// TwinCAT 3 PLC project PLC
// ProgramVersion: 3.1.4024.0
// CompilerDefines: VISU_USEWSTRING
// libraries:
//   CmpBitmapPool, * (System)
//   VisuElemBase, * (System)
//   Tc2_Standard, * (Beckhoff Automation GmbH)
//   Tc2_System, * (Beckhoff Automation GmbH)
//   Tc2_Utilities, * (Beckhoff Automation GmbH)
//   Tc3_Module, * (Beckhoff Automation GmbH)
//   VisuDialogs, * (System)
//   VisuUserMgmt, * (System)
//   VisuSymbols,3.5.10.0,System
//   VisuUserMgmt3 Interfaces,newest,System
// project tree:
//   DUTs/DUTs/DUTs/DUTs_Events/ ST_EventDefinition.TcDUT, ST_EventHistoricalSimple.TcDUT, ST_EventHistoricalSimplePersistent.TcDUT
//   DUTs/DUTs/DUTs/DUTs_HMI/ stButton.TcDUT
//   DUTs/ E_AI_Status.TcDUT, E_Mode.TcDUT
//   / GlobalTextList.TcGTLO, PlcTask.TcTTO
//   GVLs/ GVL.TcGVL, GVL_ForceMode.TcGVL, GVL_IO.TcGVL
//   GVLs/GVLs/GVLs/GVLs_Events/ GVL_EHS.TcGVL, GVL_EHSP.TcGVL, GVL_Event.TcGVL
//   GVLs/GVLs_1/ GVL_Recipe.TcGVL
//   HMI/DUTs_HMI/ stButton_1.TcDUT
//   HMI/FB/ FB_Blink_S.TcPOU, HMI.TcPOU
//   HMI/ GVL_HMI.TcGVL
//   HMI/ListyTextowe/ PrzyciskAlarmy.TcTLO, Tensometr.TcTLO, TextList_Przyciski_Menu.TcTLO
//   HMI/NEW_VISU/Frames/ E0.TcVIS, E1.TcVIS, E2.TcVIS
//   HMI/NEW_VISU/ MAIN.TcVIS, MENU_2.TcVIS, TOP.TcVIS
//   POUs/ Alarms.TcPOU, BreakthroughDetection_2.TcPOU, HydraulicPump.TcPOU, IO_Map.TcPOU, MAIN.TcPOU, Mode.TcPOU, Scaling.TcPOU, UpperPreserDrive.TcPOU, SavePresistent.TcPOU
//   POUs/FB/ FB_4_20mA_To_0_10V.TcPOU, FB_AI_Int_To_PV.TcPOU, FB_AI_mA_To_mm_Adv.TcPOU, FB_AI_Real_To_PV_Adv.TcPOU, FB_AutoManual.TcPOU, FB_Blink_S_1.TcPOU, FB_HydraulicPress_Atos_420mA.TcPOU, FB_HydraulicPumpControl.TcPOU, FB_LongPressLatch.TcPOU, FB_PositionOffset_4_20mA.TcPOU, FB_PressureToForce_PT1.TcPOU, FB_PV_To4_20mA.TcPOU, FB_RevMotorControl.TcPOU, FB_ScaleStrainGaugeForce.TcPOU, FB_ScaleTo0_10V.TcPOU, FB_ScaleTo4_20mA.TcPOU, FB_HydraulicPress_WithBreakthroughDetection_1.TcPOU
//   POUs/POUs/Events/ F_RESET_Event.TcPOU, F_SET_Event.TcPOU, P_EventHandling2.TcPOU, P_Events.TcPOU, P_EventsDefinition.TcPOU, P_EventsHandling.TcPOU, P_EventsVisu.TcPOU
//   POUs/POUs/Recipe/ RecipeManagement.TcPOU
//   VISUs/ Visualization Manager.TcVMO (not stored)
//   VISUs/VISUs/ VISU_TASK.TcTTO
// real-time tasks:
//   TASK PlcTask: cycle T#10ms, priority 20, ADS port 350
//   TASK VISU_TASK: cycle T#200000us, priority 30, ADS port 351
// I/O:
//   DEVICE Device 1 (EtherCAT) (disabled), AmsNetId 192.168.1.80.2.1
//     Term 1 (EK1818) [EK1818 EtherCAT IO-Coupler  (1A E-Bus, 8 Ch. Dig. In, 3ms, 4 Ch. Dig. Out 24V, 0,5A)]
//       Term 2 (EL4374) [EL4374 2Ch. Ana. Input, 2Ch. Ana. Output, +/-10V, +/-20mA, 16 Bit]
//       Term 6 (EL3064) [EL3064 4Ch. Ana. Input 0-10V]
//       Term 3 (EL1008) [EL1008 8Ch. Dig. Input 24V, 3ms]
//       Term 4 (EL2008) [EL2008 8Ch. Dig. Output 24V, 0.5A]
//       Term 5 (EL9011) [EL9011 End Terminal]
// variable links:
//   PLC/PLC Instance <-> Device 1 (EtherCAT)/Term 1 (EK1818)
//     PlcTask Inputs/GVL_IO.DI1_{1..8} <-> Channel {1..8}/GVL_IO.DI1_{1..8}  (8 links)
//     PlcTask Outputs/GVL_IO.DO1_{1..4} <-> Channel {9..12}/Output  (4 links)
//   PLC/PLC Instance <-> Device 1 (EtherCAT)/Term 1 (EK1818)/Term 2 (EL4374)
//     PlcTask Inputs/GVL_IO.AI_1 <-> AI Standard (Real32) Ch.1/GVL_IO.AI_1
//     PlcTask Inputs/GVL_IO.AI_2 <-> AI Standard (Real32) Ch.2/GVL_IO.AI_2
//     PlcTask Outputs/GVL_IO.AO_1 <-> AO Standard (Real32) Ch.3/GVL_IO.AO_1
//   PLC/PLC Instance <-> Device 1 (EtherCAT)/Term 1 (EK1818)/Term 3 (EL1008)
//     PlcTask Inputs/GVL_IO.DI2_{1..8} <-> Channel {1..8}/GVL_IO.DI2_{1..8}  (8 links)
//   PLC/PLC Instance <-> Device 1 (EtherCAT)/Term 1 (EK1818)/Term 4 (EL2008)
//     PlcTask Outputs/GVL_IO.DO2_{1..8} <-> Channel {1..8}/GVL_IO.DO2_{1..8}  (8 links)

CONFIGURATION PLC
    RESOURCE PLC ON TwinCAT3
        TASK PlcTask(INTERVAL := T#10ms, PRIORITY := 20);
        TASK VISU_TASK(INTERVAL := T#200000us, PRIORITY := 30);
        PROGRAM MAIN WITH PlcTask : MAIN;
        PROGRAM VisuElems_Visu_Prg WITH VISU_TASK : VisuElems.Visu_Prg;
    END_RESOURCE
END_CONFIGURATION

// ---- DUTs/DUTs/DUTs/DUTs_Events/ST_EventDefinition.TcDUT
//==================================================================================================
//							Beckhoff Automation Poland
//									23.05.2017
//	Struktura zawierajaca definicje zdarzenia
// 	v1.0	|| TC v 3.1.4020.32		|| - pierwsza wersja
//==================================================================================================
TYPE ST_EventDefinition :
STRUCT
	dwClass									: DWORD;
	dwParam									: DWORD;
	wsMessage								: WSTRING(80);
	bActive									: BOOL;	
END_STRUCT
END_TYPE

// ---- DUTs/DUTs/DUTs/DUTs_Events/ST_EventHistoricalSimple.TcDUT
//==================================================================================================
//							Beckhoff Automation Poland
//									23.05.2017
//	Struktura zawierajaca zdarzenie - pelne informacje, np. do wizualizacji
// 	v1.0	|| TC v 3.1.4020.32		|| - pierwsza wersja
//==================================================================================================
TYPE ST_EventHistoricalSimple :
STRUCT
	dwID									: DWORD;
	dwParam									: DWORD;
	dwClass									: DWORD;
	dtDateBegin								: STRING(19);//DT;
	dtDateEnd								: STRING(19);//DT;
	wsMessage								: WSTRING(80);
	dwColor									: UDINT;
END_STRUCT
END_TYPE

// ---- DUTs/DUTs/DUTs/DUTs_Events/ST_EventHistoricalSimplePersistent.TcDUT
//==================================================================================================
//							Beckhoff Automation Poland
//									23.05.2017
//	Struktura zawierajaca zane do przechowania zdarzenia w pamieci
// 	v1.0	|| TC v 3.1.4020.32		|| - pierwsza wersja
//==================================================================================================
TYPE ST_EventHistoricalSimplePersistent :
STRUCT
	dwID									: DWORD;
	dwParam									: DWORD;
	dwClass									: DWORD;
	dtDateBegin								: STRING(19);//DT;
	dtDateEnd								: STRING(19);//DT;
END_STRUCT
END_TYPE

// ---- DUTs/DUTs/DUTs/DUTs_HMI/stButton.TcDUT
TYPE stButton :
STRUCT
	{attribute 'TcEncoding':='UTF-8'}
	sName				: T_MaxString;
	bToggleCollor		: BOOL;
	bVisable			: BOOL;
	nIndexDynamicText	: UINT;
	dwColor				: DWORD;
	dwAlarmColor		: DWORD;
	
END_STRUCT
END_TYPE

// ---- DUTs/E_AI_Status.TcDUT
//{attribute 'qualified_only'}
//{attribute 'strict'}
TYPE E_AI_Status  :
(
	 AI_Status_Ok,           // wszystko w normie
    AI_Status_UnderRange,   // prąd poniżej dolnego progu (np. przerwana pętla)
    AI_Status_OverRange,    // prąd powyżej górnego progu (np. zwarcie, błąd)
    AI_Status_ConfigError   // błąd konfiguracji (InMin/InMax)
);
END_TYPE

// ---- DUTs/E_Mode.TcDUT
//{attribute 'qualified_only'}
//{attribute 'strict'}
TYPE E_Mode :
(
	Mode_Manual := 0,
    Mode_Auto   := 1
);
END_TYPE

// ---- HMI/DUTs_HMI/stButton_1.TcDUT
TYPE stButton_1 :
STRUCT
	{attribute 'TcEncoding':='UTF-8'}
	sName				: T_MaxString;
	bToggleCollor		: BOOL;
	bVisable			: BOOL;
	nIndexDynamicText	: UINT;
	dwColor				: DWORD;
	dwAlarmColor		: DWORD;
	
END_STRUCT
END_TYPE

// ---- GVLs/GVL.TcGVL
//{attribute 'qualified_only'}
VAR_GLOBAL
	AlwaysFalse					:BOOL;
	
	bControlOn					: BOOL;//kluczyk-sterowanie załączone
	bTopPreserCmdUp				: BOOL;//przycisk kolumna dociskowa do góry
	bTopPreserCmdDown			: BOOL;//przycisk kolumna dociskowa do dołu
	bCycleStartCmd				: BOOL;//przycisk start cyklu
	bCycleStopCmd				: BOOL;//przycisk stop cyklu
	bCylinderCmdUp				: BOOL;//przycisk siłownik do góry
	bCylinderCmdDown			: BOOL;//przycisk siłownik do góry
	bHydraulicUnitCmdStart		: BOOL;//przycisk agregat hydrauliczny start
	nHydraulicPressureRaw		: REAL;//ciśnienie hydrauliki-wejście analogowe
	nCylinderPositionRaw		: REAL;//pozycja siłownika-wejście analogowe
	nHydraulicPressureOut		: REAL;//cisnienie zadane na wyjscie analogowe
	bHydraulicUnitOn			: BOOL;//pottwierdzenie załączenia silnika hydrauliki z softstart
	bTopPreserClosed			: BOOL;//potwierdzenie zamknięcia docisku górnego
	bTopPreserMotorOk			: BOOL;//termik silnika docisku górnego
	bHydraulicUnitMotorOk		: BOOL;//termik silnika hydrauliki
	bHydraulicUnitCmdStop		: BOOL;//przycisk agregat hydrauliczny stop
	bOilLevelOk					: BOOL;//poziom oleju	
	bHydraulicUnitRunning       : BOOL;//softstart hydrauliki załączony
	
	bTopPreserUp				: BOOL;// wyjście -docisk górny do góry
	bTopPreserDown				: BOOL;// wyjście -docisk górny do dołu
	bHydraulicUintOn			: BOOL;// wyjście -załączenie agregatu hydraulicznego
	bLedCycleOn					: BOOL;// wyjście -LED cykl załączony
	bReliefValveOn				: BOOL;// wyjście -zawór odciążający załączony
	bCylinderValveUp			: BOOL;// wyjście -zawór siłownik do góry
	bCylinderValveDown			: BOOL;// wyjście -zawór siłownik do dołu
	bProportionalValveEnable	: BOOL;// wyjście -zawór proporcjonalny załączony	
	bLedHydraulicUnitOn			: BOOL;// wyjście -LED hydraulika załączona
	
	
	

	nHydraulicPressureOut0_10V: LREAL;
END_VAR

// ---- GVLs/GVLs/GVLs/GVLs_Events/GVL_EHS.TcGVL
//==================================================================================================
//							Beckhoff Automation Poland
//									23.05.2017
// 	v1.0	|| TC v 3.1.4020.32		|| - pierwsza wersja
//==================================================================================================
{attribute 'qualified_only'}
VAR_GLOBAL CONSTANT
	diEventsDefinition						: UDINT 	:= 1000;				// Rozmiar tablicy definicji zdarzen, powinna byc w zakresie 5..1000
	diNoOfEvents							: UDINT 	:= 1000;				// Rozmiar tablicy zdarzen historycznych, powinna byc w zakresie 5..1000
END_VAR
VAR_GLOBAL
	stActTime								: TIMESTRUCT;				// Aktualny czas sytemowy w formie struktury
	dtActTime								: STRING(19);//DT;						// Aktualny czas sytemowy
	arrEventDefinition 						: ARRAY [1..GVL_EHS.diEventsDefinition] OF ST_EventDefinition;
	arrEventVisu							: ARRAY [1..GVL_EHS.diNoOfEvents] OF ST_EventHistoricalSimple;		// Pokazywane na wizualizacji - po filtracji
	dwLanguageId							: DWORD := 1045;			// Kod jezyka wyswietlania - Microsoft Locale ID Values
END_VAR

// ---- GVLs/GVLs/GVLs/GVLs_Events/GVL_EHSP.TcGVL
//==================================================================================================
//							Beckhoff Automation Poland
//									23.05.2017
// 	v1.0	|| TC v 3.1.4020.32		|| - pierwsza wersja
//==================================================================================================
{attribute 'qualified_only'}
VAR_GLOBAL PERSISTENT
	arrEvent								: ARRAY [1..GVL_EHS.diNoOfEvents] OF ST_EventHistoricalSimplePersistent;
END_VAR

// ---- GVLs/GVLs/GVLs/GVLs_Events/GVL_Event.TcGVL
{attribute 'qualified_only'}
VAR_GLOBAL
	bAlarm :BOOL;
	bWarning:BOOL;
	bMessage:BOOL;
	aAlarm: ARRAY[0..100] OF BOOL;
	aWarning: ARRAY[0..100] OF BOOL;
	aMessage: ARRAY[0..100] OF BOOL;
	bJestAalrm: BOOL;
	bFilterActiveOnly2: BOOL;
	bJestOstrzezenie: BOOL;
	bJestAalrmLekki: BOOL;
END_VAR

// ---- GVLs/GVLs_1/GVL_Recipe.TcGVL
{attribute 'qualified_only'}
VAR_GLOBAL CONSTANT
	cMaxTableRows 			: INT := 30;

END_VAR
VAR_GLOBAL
	// zmienne receptury
	(*Zmienna1				: LREAL;
	Zmienna2				: LREAL;
	Zmienna3				: LREAL;
	Zmienna4				: LREAL;
	Zmienna5				: INT;
	Zmienna6				: INT;
	Zmienna7				: LREAL;
	Zmienna8				: LREAL;
	Zmienna9				: LREAL;
	Zmienna10				: LREAL;
	*)
	// zmienne do obslugi
	nRecipeCount			: INT;
	aRecipeNames 			: ARRAY[0..cMaxTableRows] OF STRING;
	aVariableNames 			: ARRAY[0..cMaxTableRows] OF STRING;
	aVariableValues 		: ARRAY[0..cMaxTableRows] OF STRING;
	nRecipeIndex			: INT;
	nRecipeSelectionIndex	: INT;
	nVariableIndex			: INT;
	aCurrentValues			: ARRAY[0..cMaxTableRows] OF LREAL;
	


	bZapiszParametry: BOOL;
	bCzytajParametry: BOOL;
	nRecipeSelectionIndexTemp: INT;
	
END_VAR

// ---- GVLs/GVL_ForceMode.TcGVL
{attribute 'qualified_only'}
VAR_GLOBAL
(* ===== Przełączniki =====
	   bModeForce:        FALSE = regulacja i przebicie od ciśnienia (jak dotychczas)
	                      TRUE  = regulacja i przebicie od siły
	   bForceRange100t:   FALSE = tensometr 50 t  (2,5 V = 50 t)
	                      TRUE  = tensometr 100 t (2,5 V = 100 t)
	   Oba można podpiąć pod przełącznik na pulpicie albo pod HMI.
	   Domyślnie FALSE, więc po wgraniu maszyna zostaje w trybie ciśnienia, zakres 50 t.
	*)
	bModeForce					: BOOL := FALSE;
	bForceRange100t				: BOOL := FALSE;

	(* ===== Drugi setpoint — siła [t] =====
	   Odpowiednik setpointów ciśnienia. Używane tylko w trybie siły.
	   Wartość wpisana powyżej wybranego zakresu jest obcinana (patrz *_Eff).
	*)
	nForceSetpointManual		: REAL := 0.0;	(* t, tryb ręczny *)
	nForceSetpointAutoMin		: REAL := 0.0;	(* t, auto *)
	nForceSetpointAutoMax		: REAL := 0.0;	(* t, auto *)
	nBreakDeltaForce			: REAL := 0.0;	(* t, spadek siły w oknie czasu = przebicie *)

	(* ===== Pomiar =====
	   Powiąż nForceInput_V z kanałem AI 0–10 V. Jednostka: wolty (0.0 … 10.0).
	   Zakres roboczy przetwornika to 0.0 … 2.5 V. Powyżej 2.55 V = błąd zakresu.
	*)
	nForceInput_V				: REAL := 0.0;

	nForce_t					: REAL;	(* wartość chwilowa, t *)
	nForce_kg					: REAL;	(* kgf *)
	nForce_N					: REAL;
	nForce_kN					: REAL;
	nForce_pct					: REAL;	(* % wybranego zakresu *)
	nForceFullScale_t			: REAL;	(* 50 albo 100 *)
	bForceSensorOk				: BOOL;
	bForceOverrange				: BOOL;
	bForceUnderrange			: BOOL;

	nForce_Target				: REAL;	(* bieżące zadanie siły w trybie siły [t]; 0 w trybie ciśnienia *)

	

	(* Setpointy faktycznie podane do regulatora po obcięciu do zakresu. *)
	nForceSetpointManual_Eff	: REAL;
	nForceSetpointAutoMin_Eff	: REAL;
	nForceSetpointAutoMax_Eff	: REAL;
	nBreakDeltaForce_Eff		: REAL;
	bForceSetpointLimited		: BOOL;	(* wpisana wartość była poza 0 … pełny zakres albo delta < 0 *)
	bForceCfgFault				: BOOL;	(* AutoMin > AutoMax po obcięciu *)
	bForceInhibit				: BOOL;	(* tryb siły i zły tensometr — ruch w górę jest zablokowany, dół zostaje *)
	bMotionHold					: BOOL;	(* zmiana trybu lub zakresu 50/100 t w ruchu — puść przyciski *)
	bRegulatorActive			: BOOL;
	bAlarm						: BOOL;
	nActiveSetpointManual		: REAL;	(* to, co w tym cyklu poszło jako setpoint ręczny: bar albo t *)
	nActiveActual				: REAL;	(* to, co w tym cyklu poszło jako wartość rzeczywista *)
END_VAR

// ---- GVLs/GVL_IO.TcGVL
//{attribute 'qualified_only'}
VAR_GLOBAL
//---------------------------------------------	
// EK 1818

	DI1_1 AT %I*: BOOL;
	DI1_2 AT %I*: BOOL;
	DI1_3 AT %I*: BOOL;
	DI1_4 AT %I*: BOOL;
	DI1_5 AT %I*: BOOL;
	DI1_6 AT %I*: BOOL;
	DI1_7 AT %I*: BOOL;
	DI1_8 AT %I*: BOOL;
	
	DO1_1 AT %Q*: BOOL;
	DO1_2 AT %Q*: BOOL;
	DO1_3 AT %Q*: BOOL;
	DO1_4 AT %Q*: BOOL;
//--------------------------------------------	
// EL 4374	
	AI_1 AT %I*: REAL;
	AI_2 AT %I*: REAL;
	AO_1 AT %Q*: REAL;
	AO_2 AT %Q*: REAL;
//--------------------------------------------
// EL 1008	
	DI2_1 AT %I*: BOOL;
	DI2_2 AT %I*: BOOL;
	DI2_3 AT %I*: BOOL;
	DI2_4 AT %I*: BOOL;
	DI2_5 AT %I*: BOOL;
	DI2_6 AT %I*: BOOL;
	DI2_7 AT %I*: BOOL;
	DI2_8 AT %I*: BOOL;
	
//--------------------------------------------
//EL 2008
	DO2_1 AT %Q*: BOOL;
	DO2_2 AT %Q*: BOOL;
	DO2_3 AT %Q*: BOOL;
	DO2_4 AT %Q*: BOOL;
	DO2_5 AT %Q*: BOOL;
	DO2_6 AT %Q*: BOOL;
	DO2_7 AT %Q*: BOOL;
	DO2_8 AT %Q*: BOOL;
	// sygnał z przekaźnika bezpieczeństwa
	bEstopOk: BOOL;
END_VAR

// ---- HMI/GVL_HMI.TcGVL
{attribute 'qualified_only'}
VAR_GLOBAL
	hmiPanel	: HMI;
	
	bKlodka: BOOL;
	bResetAlarm: BOOL;
	
	tBreak_Time_Window: TIME;
	sMode: STRING;
	nPressBreak: REAL;
	nPositionBreak: REAL;
	nPressStart: REAL;
	nPositionStart: REAL;
	Force_N: REAL;
	Force_kg: REAL;
	Force_kg_2: REAL;
	Force_N_2: REAL;
	(* Zatrzask w chwili wykrycia przebicia — pomiar z tensometru, niezależnie od trybu. *)
	nForce_t_Break				: REAL;
	nForce_kg_Break				: REAL;
	nForce_N_Break				: REAL;
	nForce_kN_Break				: REAL;
END_VAR
VAR_GLOBAL PERSISTENT
	nBreak_Time_Window			: INT;
	nPressureSetpointManual: REAL;
	nBreakDeltaPress: REAL;
	nBreakDeltaPos: REAL;
	PressureSetpointAutoMin: LREAL;
	PressureSetpointAutoMax: LREAL;
	// czas rampy Auto[ms]
	nRamp_Time: DINT:=120;
END_VAR
VAR_GLOBAL CONSTANT
	// Czasem w HMI trzeba podać kolor w wersji 16 
	dwRed				: DWORD  := 16#FFE62545;
	dwGreen				: DWORD  := 16#FF007D00;
	dwYelow				: DWORD  := 16#FFFFFF00;
	dwBlack				: DWORD  := 16#FF000000;
	dwGrey_B			: DWORD  := 16#FF636363;
	dwGrey_W			: DWORD  := 16#FFC8C8C8;
	dwWhite				: DWORD  := 16#FFFFFFFF;
	dwBackGround		: DWORD	 := 16#FFABA494;
	
END_VAR

// ---- POUs/MAIN.TcPOU
PROGRAM MAIN
VAR
END_VAR

GVL_HMI.hmiPanel();

UpperPreserDrive();
HydraulicPump();
BreakthroughDetection_2();



P_Events();
P_EventsDefinition();
Alarms();
Scaling();
SavePresistent();
Mode();
IO_Map();

END_PROGRAM

// ---- POUs/UpperPreserDrive.TcPOU
PROGRAM UpperPreserDrive
VAR
	fbUupperPreser: FB_RevMotorControl;
	
	bStop: BOOL;
	
END_VAR

fbUupperPreser(
	bForward:=.bTopPreserCmdDown , 
	bReverse:=.bTopPreserCmdUp , 
	bStop:=bStop , 
	bThermalOk:=.bTopPreserMotorOk , 
	bLimitSwitchFwd:=TRUE , 
	bLimitSwitchRev:=.bTopPreserClosed , 
	bEmergencyStop:=.bEstopOk , 
	bEnable:=bControlOn , 
	bRunForward=>.bTopPreserDown , 
	bRunReverse=>.bTopPreserUp , 
	bRunning=> , 
	bFault=> , 
	bReady=> );

END_PROGRAM

// ---- POUs/FB/FB_RevMotorControl.TcPOU
FUNCTION_BLOCK FB_RevMotorControl
VAR_INPUT
    bForward            : BOOL;  // Komenda jazdy w przód
    bReverse            : BOOL;  // Komenda jazdy w tył
    bStop               : BOOL := FALSE;  // Zatrzymanie ręczne (opcjonalne)
    bThermalOk          : BOOL := TRUE;   // Termik silnika OK (NC → 0 = zadziałany)
    bLimitSwitchFwd     : BOOL := TRUE;   // Krańcówka przód (NC → 0 = osiągnięta)
    bLimitSwitchRev     : BOOL := TRUE;   // Krańcówka tył  (NC → 0 = osiągnięta)
    bEmergencyStop      : BOOL := TRUE;   // E-Stop (NC → 0 = wciśnięty)
    bEnable             : BOOL := TRUE;   // Zewnętrzne zezwolenie
END_VAR

VAR_OUTPUT
    bRunForward         : BOOL;  // Stycznik – jazda w przód
    bRunReverse         : BOOL;  // Stycznik – jazda w tył
    bRunning            : BOOL;  // Silnik pracuje (którykolwiek kierunek)
    bFault              : BOOL;  // Błąd wymagający kasowania (głównie termik)
    bReady              : BOOL;  // System gotowy do pracy
END_VAR

VAR
    bIntForward         : BOOL := FALSE;  // Wewnętrzny stan przód
    bIntReverse         : BOOL := FALSE;  // Wewnętrzny stan tył
    bThermalFault       : BOOL := FALSE;  // Ręczna pamięć błędu termicznego (zamiast SR)
    tAntiTieDelay1       : TON;            // Opóźnienie przeciwzwarciowe 400 ms
	tAntiTieDelay2       : TON;            // Opóźnienie przeciwzwarciowe 400 ms
    bFirstCycle         : BOOL := TRUE;
END_VAR



//===================================================================
// Poprawiona logika – krańcówki działają prawidłowo!
//===================================================================

IF bFirstCycle THEN
  
    tAntiTieDelay1.PT := T#300MS;
	tAntiTieDelay2.PT := T#300MS;
	  bFirstCycle := FALSE;
END_IF;

// 1. Natychmiastowe wyłączenie przy braku bezpieczeństwa
IF NOT bEmergencyStop OR NOT bThermalOk THEN
    bIntForward := FALSE;
    bIntReverse := FALSE;
END_IF;

// 2. Ręczna pamięć błędu termicznego
IF NOT bThermalOk AND bRunForward AND bRunReverse THEN
    bThermalFault := TRUE;                    // SET
END_IF;
IF bEmergencyStop AND bThermalOk AND (bStop OR (bForward AND bReverse)) THEN
    bThermalFault := FALSE;                   // RST
END_IF;

// 3. Główna logika kierunku – KRAŃCÓWKI TYLKO BLOKUJĄ SWÓJ KIERUNEK!
IF NOT bThermalFault AND bEnable AND bEmergencyStop AND bThermalOk THEN

    // Żądanie jazdy w przód – dozwolone tylko jeśli krańcówka przód jest zwolniona
    IF bForward AND NOT bReverse AND bLimitSwitchFwd AND NOT bIntReverse THEN
        bIntForward := TRUE;
    ELSIF NOT bLimitSwitchFwd OR bReverse THEN
        bIntForward := FALSE;                 // krańcówka przód osiągnięta → wyłącz przód
    END_IF;

    // Żądanie jazdy w tył – dozwolone tylko jeśli krańcówka tył jest zwolniona
    IF bReverse AND NOT bForward AND bLimitSwitchRev and not bIntForward THEN
        bIntReverse := TRUE;
    ELSIF NOT bLimitSwitchRev OR bForward THEN
        bIntReverse := FALSE;                 // krańcówka tył osiągnięta → wyłącz tył
    END_IF;

    // Zatrzymanie ręczne lub brak komendy
    IF bStop OR (NOT bForward AND NOT bReverse)OR (bForward AND  bReverse) THEN
        bIntForward := FALSE;
        bIntReverse := FALSE;
    END_IF;

END_IF;

// 4. Opóźnienie przeciwzwarciowe 400 ms
tAntiTieDelay1(IN := bForward );

IF tAntiTieDelay1.Q THEN
    bRunForward := bIntForward;
    
ELSE
    bRunForward := FALSE;
   
END_IF;

tAntiTieDelay2(IN := bReverse);

IF tAntiTieDelay2.Q THEN
   
    bRunReverse := bIntReverse;
ELSE
   
    bRunReverse := FALSE;
END_IF;
// 5. Wyjścia diagnostyczne
bRunning := bRunForward OR bRunReverse;

bReady   := bEmergencyStop
            AND bThermalOk
            AND bEnable
            AND NOT bThermalFault;

bFault   := bThermalFault;

END_FUNCTION_BLOCK

// ---- POUs/HydraulicPump.TcPOU
PROGRAM HydraulicPump
VAR
    
	fbHydPump: FB_HydraulicPumpControl;
	
	bMaxPressure: BOOL;
	
	fbBlink: FB_Blink_S_1;
END_VAR

fbHydPump(
	bStart         := bHydraulicUnitCmdStart,
    bStop          := bHydraulicUnitCmdStop AND NOT.bCylinderCmdDown,
    bEmergencyStop := bEStopOk,          // NC – 0=wciśnięty
    bThermalOk     := bHydraulicUnitMotorOk,        // NC – 0=zadziałany
    bPressureOk    := NOT bMaxPressure,   // czujnik NO → inwertujemy
	bOilLevel	   := TRUE,
    bEnable        := bControlOn,
	bPumpRun=> bLedHydraulicUnitOn, 
	bRunning=>.bHydraulicUintOn , 
	bFault=> , 
	bReady=> , 
	bFaultThermal=> , 
	bFaultPressure=> );
(*
Q_PumpContactor := HydPump.bPumpRun;
HMI_Alarm       := HydPump.bFault;
HMI_Ready       := HydPump.bReady;
HMI_ThermalErr  := HydPump.bFaultThermal;
HMI_PressureErr := HydPump.bFaultPressure;
*)

//=======================================================================
//			MAX. CIŚNIENIE
bMaxPressure:=Scaling.PressureAI.PV_Value>390;
//=======================================================================
//		ENABLE NA ZAWÓR PROPORCJONlNY
bProportionalValveEnable:= .bEstopOk AND (bCylinderValveUp or bCylinderValveDown);
//=======================================================================
//			LED HYDRAULIKA ZAŁACZONA
fbBlink(Tv:=T#400MS , Q=> );

IF bHydraulicUintOn THEN
 IF NOT bHydraulicUnitRunning THEN
	bLedHydraulicUnitOn:=fbBlink.Q;
	ELSIF
		 bHydraulicUnitRunning THEN
		 bLedHydraulicUnitOn:=bHydraulicUintOn;
		
	END_IF	
	ELSE
			bLedHydraulicUnitOn:=FALSE;
END_IF
//=========================================================================

END_PROGRAM

// ---- POUs/FB/FB_HydraulicPumpControl.TcPOU
FUNCTION_BLOCK FB_HydraulicPumpControl
// Sterowanie pompą hydrauliczną – 
VAR_INPUT
    bStart          : BOOL;  // Przycisk START (impulsowy lub podtrzymany)
    bStop           : BOOL;  // Przycisk STOP
    bEmergencyStop  : BOOL := TRUE;   // E-Stop (NC → 0 = wciśnięty)
    bThermalOk      : BOOL := TRUE;   // Zabezpieczenie termiczne silnika (NC → 0 = zadziałane)
    bPressureOk     : BOOL := TRUE;   // Czujnik ciśnienia – OK gdy NIE ma nadciśnienia (NO → 1 = za wysokie → po inwersji)
	bOilLevel		: BOOL := TRUE;	  // Czujnik poziomu oleju OK=1
    bEnable         : BOOL := TRUE;   // Zewnętrzne zezwolenie na pracę (np. tryb auto)
END_VAR

VAR_OUTPUT
    bPumpRun        : BOOL;  // Wyjście na stycznik pompy
    bRunning        : BOOL;  // Pompa aktualnie pracuje
    bFault          : BOOL;  // Błąd wymagający kasowania (termik lub nadciśnienie)
    bReady          : BOOL;  // Wszystko sprawne i gotowe do startu
    bFaultThermal   : BOOL;  // Szczegółowy powód błędu – termik
    bFaultPressure  : BOOL;  // Szczegółowy powód błędu – nadciśnienie
END_VAR

VAR
    bInternalRun    : BOOL := FALSE;     // Wewnętrzny stan pracy (z pamięcią)
    bFaultLatched   : BOOL := FALSE;     // Ręczny latch na błąd (zamiast SR)
    bSafetyOk       : BOOL;              // Aktualny stan bezpieczeństwa
    bFirstCycle     : BOOL := TRUE;
END_VAR

//===================================================================
// Główna logika sterowania pompą – 
//===================================================================

IF bFirstCycle THEN
    bFirstCycle := FALSE;
END_IF;

// 1. Aktualny stan bezpieczeństwa (musi być spełniony w każdej chwili)
bSafetyOk := bEmergencyStop          // E-Stop zwolniony
             AND bThermalOk          // Termik nie zadziałał
             AND bPressureOk         // Ciśnienie w normie
             AND bEnable            // Zewnętrzne zezwolenie
			AND bOilLevel;
// 2. Ręczny latch błędu (zapamiętujemy tylko termik, poziom i nadciśnienie)
IF NOT bSafetyOk AND (NOT bThermalOk OR NOT bOilLevel OR NOT bPressureOk) THEN
    bFaultLatched := TRUE;                       // SET – zapamiętaj błąd
END_IF;

IF bSafetyOk AND (bStart OR NOT bStop) THEN
    bFaultLatched := FALSE;                      // RST – kasowanie po potwierdzeniu
END_IF;

// 3. Natychmiastowe wyłączenie przy braku bezpieczeństwa
IF NOT bSafetyOk THEN
    bInternalRun := FALSE;
END_IF;

// 4. Logika ręcznego start/stop (działa tylko gdy nie ma zapamiętanego błędu)
IF NOT bFaultLatched AND bSafetyOk THEN
    IF bStart AND NOT NOT bStop THEN
        bInternalRun := TRUE;                    // Start ma przewagę nad Stop
    ELSIF NOT bStop THEN
        bInternalRun := FALSE;
    END_IF;
END_IF;

// 5. Wyjścia końcowe
bPumpRun   := bInternalRun AND bSafetyOk;        // Ostateczne wyjście na stycznik
bRunning   := bPumpRun;

bReady     := bSafetyOk AND NOT bFaultLatched;   // Zielone światło na HMI

bFault     := bFaultLatched OR NOT bEmergencyStop;  // Stały alarm przy błędzie lub E-Stop

// 6. Szczegółowe przyczyny błędu (bardzo przydatne na HMI)
bFaultThermal   := bFaultLatched AND NOT bThermalOk;
bFaultPressure  := bFaultLatched AND NOT bPressureOk;

END_FUNCTION_BLOCK

// ---- POUs/FB/FB_Blink_S_1.TcPOU
(********************************************************************************************)
(*							Beckhoff Automation Poland										*)
(*								FB_Blink_S	 v1.1											*)
(*									9.11.2007												*)
(*						Blok funkcyjny zegara synchronicznego								*)
(*__________________________________________________________________________________________*)

FUNCTION_BLOCK FB_Blink_S_1
VAR_INPUT
	Tv										:	TIME;				(*Czas trwania impulsu i przerwy*)
END_VAR
VAR_OUTPUT
	Q										:	BOOL;				(*Wyjscie*)
END_VAR
VAR
	ton1									:	TON;
	ton2									:	TON;
END_VAR

ton1(IN:= NOT ton2.Q, PT:=Tv);
Q:=ton1.Q;
ton2(IN:=ton1.Q , PT:=ton1.PT );

END_FUNCTION_BLOCK

// ---- POUs/Scaling.TcPOU
PROGRAM Scaling
VAR
	AI_PressureRaw   : REAL;
    PressureAI  : FB_AI_Real_To_PV_Adv;
	AI_PositionRaw: REAL;
	PositionAI  : FB_AI_Real_To_PV_Adv;
///////////////////////////////////////////////
	AI_Raw  : INT;                      // np. wartość z karty
    fbPresureTo4_20 : FB_ScaleTo4_20mA;
	fbPresureToPV  : FB_AI_Int_To_PV;
	fbPositionTo4_20 : FB_ScaleTo4_20mA;
	fbPositionToPV  : FB_AI_Int_To_PV;
    Current : REAL;
	
	nCurrentPressure_4_20mA: REAL;
	nCurrentPressure_bar: REAL;
	nCurrentPressure_PC: REAL;
	nCurrentPosition_4_20mA: REAL;
	nCurrentPosition_mm: REAL;
	nCurrentPosition_PC: REAL;
	
	fbPressureMax: FB_PV_To4_20mA;
	
	fbPressureMin: FB_PV_To4_20mA;
	////////////////////////////////////////////////////
	

    AI_mA     : REAL;  (* tu wstaw wartość z kanału AI w mA *)
    BtnZero   : BOOL;  (* przycisk zerowania *)

    PosRaw    : REAL;
    PosZero   : REAL;
	
	fbPressureToForce: FB_PressureToForce_PT1;
	fbForceRawToForceVolt: FB_ScaleTo0_10V;
	fbFB_ScaleTo0_10V: FB_ScaleTo0_10V;
END_VAR
	
VAR PERSISTENT
	fbPos : FB_PositionOffset_4_20mA;
END_VAR

(*
//============================================================
//		SKALOWANIE CIŚNIENIA
//------------------------------------------------------------
//		AI to 4-20mA
AI_Raw := iHydraulicPressureRaw;  //  wartość z wejścia

fbPresureTo4_20(
    InRaw := AI_Raw,
    InMin := 0,
    InMax := 32767
);


nCurrentPressure_4_20mA := fbPresureTo4_20.Out_mA;  // wynik w mA (4–20)
//-------------------------------------------------------------
//			AI to bar
fbPresureToPV(
    InRaw  := AI_Raw,
    InMin  := 0,
    InMax  := 32767,
    PV_Min := 0.0,     // 0 bar
    PV_Max := 400.0     // 400 bar
);

nCurrentPressure_bar :=fbPresureToPV.PV_Value;//  → ciśnienie [bar]
nCurrentPressure_PC :=fbPresureToPV.PV_Percent; //→ [% zakresu]

//=================================================================
//			SKALOWANIE POZYCJI
//-----------------------------------------------------------------
//			AI to 4-20mA
AI_Raw := iCylinderPositionRaw;  //  wartość z wejścia

fbPositionTo4_20(
    InRaw := AI_Raw,
    InMin := 0,
    InMax := 32767
);


nCurrentPosition_4_20mA := fbPositionTo4_20.Out_mA;  // wynik w mA (4–20)
//-------------------------------------------------------------
//			AI to mm
fbPositionToPV(
    InRaw  := AI_Raw,
    InMin  := 0,
    InMax  := 32767,
    PV_Min := 0.0,     // 0 mm
    PV_Max := 100.0     // 100 mm
);

nCurrentPosition_mm :=fbPositionToPV.PV_Value;//  → pozycja [mm]
nCurrentPosition_PC :=fbPositionToPV.PV_Percent; //→ [% zakresu]
*)
/////////////////////////////////////////////////////////////////////

//============================================================
//		SKALOWANIE CIŚNIENIA
//------------------------------------------------------------

AI_PressureRaw:=nHydraulicPressureRaw*1000 ;

PressureAI(
    InRaw       := AI_PressureRaw,
    InMin       := 4.0,
    InMax       := 20.0,
    PV_Min      := 0.0,    // 0 bar
    PV_Max      := 400.0,   // 400 bar
    LowLimit_mA := 3.6,
    HighLimit_mA:= 21.0
);

// Wyniki:
 PressureAI.Out_mA ;     //→ prąd pętli [mA]
 PressureAI.PV_Value;    //→ ciśnienie [bar]
 PressureAI.PV_Percent;  //→ % zakresu (0..100)
 PressureAI.Status;      //→ OK / UnderRange / OverRange / ConfigError
 PressureAI.Valid ;      //→ TRUE tylko gdy OK

//============================================================
//		SKALOWANIE POZYCJI
//------------------------------------------------------------

AI_PositionRaw:=nCylinderPositionRaw*1000 ;
(*
PositionAI(
    InRaw       := AI_PositionRaw,
    InMin       := 4.0,
    InMax       := 20.0,
    PV_Min      := 0.0,    // 0 bar
    PV_Max      := 125.0,   // 125 mm
    LowLimit_mA := 3.6,
    HighLimit_mA:= 21.0
);

// Wyniki:
 PositionAI.Out_mA ;     //→ prąd pętli [mA]
 PositionAI.PV_Value;    //→ pozycja [mm]
 PositionAI.PV_Percent;  //→ % zakresu (0..100)
 PositionAI.Status;      //→ OK / UnderRange / OverRange / ConfigError
 PositionAI.Valid ;      //→ TRUE tylko gdy OK
*)

fbPos(
    Enable  := TRUE,
    In_mA   := AI_PositionRaw,
    SetZero := fbPos.SetZero,
    Range_mm := 125.0
);


 //==================================================================
 // SKALOWANIE CIŚNIEŃ ZADANYCH 
 
 fbPressureMax(
	PV:=GVL_HMI.PressureSetpointAutoMax , 
	PV_Min:=0 , 
	PV_Max:= 400, 
	ClampOutput:= , 
	I_mA=> , 
	Error=> );
	
 //==================================================================
 // SKALOWANIE CIŚNIEŃ ZADANYCH 
 
 fbPressureMin(
	PV:=GVL_HMI.PressureSetpointAutoMin , 
	PV_Min:=0 , 
	PV_Max:= 400, 
	ClampOutput:= , 
	I_mA=> , 
	Error=> );	
//===================================================================
//		PRZELICZENIE CISNIENIA NA SIŁĘ
fbPressureToForce(
	Pressure_bar:=PressureAI.PV_Value , 
	PistonDiam_m:=0.45 , 
	Efficiency:=0.9 , 
	FilterTime_s:= 0.01, 
	CycleTime_s:=0.01 , 
	EnableFilter:=TRUE , 
	Force_N=>GVL_HMI.Force_N , 
	ForceRaw_N=> ,
	Force_kg =>GVL_HMI.Force_kg,
    ForceRaw_kg=>);
//===================================================================
//		SKALOWANIE WEJŚCIA 0-10V NA vOLTY
fbFB_ScaleTo0_10V(
	InRaw:=IO_Map.AI3 , 
	InMin:=0 , 
	InMax:=32767 , 
	Out_V=>GVL_ForceMode.nForceInput_V , 
	OutPercent=> , 
	Error=> );

END_PROGRAM

// ---- POUs/FB/FB_AI_Real_To_PV_Adv.TcPOU
FUNCTION_BLOCK FB_AI_Real_To_PV_Adv
VAR_INPUT
    // Wejście z karty (skalowane, typu REAL)
    InRaw        : REAL;        // wartość z przetwornika A/D jako REAL
    InMin        : REAL := 0.0; // dolna granica (np. 0.0)
    InMax        : REAL := 32767.0; // górna granica (np. 32767.0)

    // Zakres procesu (jednostki fizyczne)
    PV_Min       : REAL;       // np. 0.0 bar
    PV_Max       : REAL;       // np. 10.0 bar

    // Progi diagnostyczne pętli prądowej
    LowLimit_mA  : REAL := 3.6;  // poniżej → Underrange
    HighLimit_mA : REAL := 21.0; // powyżej → Overrange
END_VAR

VAR_OUTPUT
    Out_mA       : REAL;       // wyliczony prąd mA (bez ograniczania)
    PV_Value     : REAL;       // wartość procesowa w jednostkach fizycznych
    PV_Percent   : REAL;       // 0–100 % zakresu (po zacięciu do 0..100%)
    Status       : E_AI_Status;// OK / Underrange / Overrange / ConfigError
    Valid        : BOOL;       // TRUE gdy Status = OK
END_VAR

VAR
    ratioRaw, ratioClamped : REAL;
END_VAR

// ---- Sprawdzenie poprawności konfiguracji zakresu wejścia ----
IF InMax <= InMin THEN
    // Błąd konfiguracji – nie liczymy nic więcej
    Status     := AI_Status_ConfigError;
    Valid      := FALSE;
    Out_mA     := 4.0;
    PV_Value   := PV_Min;
    PV_Percent := 0.0;
ELSE
    // ---- Krok 1: REAL → udział 0..1 (jeszcze bez ograniczania) ----
    ratioRaw := (InRaw - InMin) / (InMax - InMin);

    // ---- Krok 2: udział → prąd 4–20 mA (bez ograniczania) ----
    Out_mA := 4.0 + ratioRaw * 16.0;  // 4..20 mA dla ratio 0..1

    // ---- Diagnostyka pętli prądowej na "surowym" Out_mA ----
    IF Out_mA < LowLimit_mA THEN
        Status := AI_Status_UnderRange;
        Valid  := FALSE;
    ELSIF Out_mA > HighLimit_mA THEN
        Status := AI_Status_OverRange;
        Valid  := FALSE;
    ELSE
        Status := AI_Status_Ok;
        Valid  := TRUE;
    END_IF;

    // ---- Krok 3: zacięcie udziału do 0..1 do dalszego przeliczania PV ----
    ratioClamped := ratioRaw;
    IF ratioClamped < 0.0 THEN ratioClamped := 0.0; END_IF;
    IF ratioClamped > 1.0 THEN ratioClamped := 1.0; END_IF;

    // ---- Krok 4: udział 0..1 → jednostki fizyczne ----
    PV_Value   := PV_Min + ratioClamped * (PV_Max - PV_Min);
    PV_Percent := ratioClamped * 100.0;
END_IF;

END_FUNCTION_BLOCK

// ---- POUs/FB/FB_ScaleTo4_20mA.TcPOU
FUNCTION_BLOCK FB_ScaleTo4_20mA

VAR_INPUT
    InRaw      : INT;    // Sygnał z wejścia analogowego (INT)
    InMin      : INT;    // Dolna granica (np. 0)
    InMax      : INT;    // Górna granica (np. 32767)
END_VAR

VAR_OUTPUT
    Out_mA     : REAL;  // Wyjście 4–20 mA
    OutPercent : REAL;  // Procent 0–100%
    Error      : BOOL;  // Błąd zakresu
END_VAR

VAR
    scaled : REAL;
END_VAR

// Zabezpieczenie przed dzieleniem przez zero
IF InMax <= InMin THEN
    Out_mA := 4.0;
    OutPercent := 0.0;
    Error := TRUE;
ELSE
    Error := FALSE;

    // Konwersja INT → REAL i skalowanie do 0–1
    scaled := (INT_TO_REAL(InRaw - InMin)) / INT_TO_REAL(InMax - InMin);

    // Ograniczenie do 0…1
    IF scaled < 0.0 THEN scaled := 0.0; END_IF;
    IF scaled > 1.0 THEN scaled := 1.0; END_IF;

    OutPercent := scaled * 100.0;

    // Skala na 4–20 mA
    Out_mA := 4.0 + (scaled * 16.0);
END_IF;

END_FUNCTION_BLOCK

// ---- POUs/FB/FB_AI_Int_To_PV.TcPOU
FUNCTION_BLOCK FB_AI_Int_To_PV
VAR_INPUT
    InRaw    : INT;   // z karty
    InMin    : INT;   // np. 0
    InMax    : INT;   // np. 32767

    PV_Min   : REAL;  // np. 0.0 bar
    PV_Max   : REAL;  // np. 10.0 bar
END_VAR

VAR_OUTPUT
    PV_Value   : REAL;  // w jednostkach fizycznych
    PV_Percent : REAL;  // 0–100 %
    ErrorConfig: BOOL;
END_VAR

VAR
    ratio   : LREAL;
    pv      : LREAL;
END_VAR

IF InMax <= InMin THEN
    ErrorConfig := TRUE;
    PV_Value    := PV_Min;
    PV_Percent  := 0.0;
ELSE
    ErrorConfig := FALSE;

    // 0..1
    ratio := (INT_TO_LREAL(InRaw) - INT_TO_LREAL(InMin)) / (INT_TO_LREAL(InMax) - INT_TO_LREAL(InMin));
    IF ratio < 0.0 THEN ratio := 0.0; END_IF;
    IF ratio > 1.0 THEN ratio := 1.0; END_IF;

    // do PV_Min..PV_Max
    pv        := (PV_Min) + ratio * ((PV_Max) - (PV_Min));
    PV_Value  := (*INT_TO_REAL*)(pv);
    PV_Percent:= LREAL_TO_REAL(ratio * 100.0);
END_IF;

END_FUNCTION_BLOCK

// ---- POUs/FB/FB_PV_To4_20mA.TcPOU
FUNCTION_BLOCK FB_PV_To4_20mA
VAR_INPUT
    PV           : LREAL; (* aktualne ciśnienie, np. [bar] *)
    PV_Min       : LREAL; (* dolny zakres przetwornika *)
    PV_Max       : LREAL; (* górny zakres przetwornika *)
    ClampOutput  : BOOL;  (* jeżeli TRUE – ograniczaj do zakresu 4–20 mA *)
END_VAR

VAR_OUTPUT
    I_mA    : LREAL; (* wyjście prądowe w mA *)
    Error   : BOOL;  (* TRUE gdy PV_Min >= PV_Max *)
END_VAR

VAR
    spanPV  : LREAL;
    spanI   : LREAL := 16.0; (* 20 mA - 4 mA *)
    tmpI    : LREAL;
END_VAR

(* --------------------------------------------- *)
(* Konwersja PV -> 4–20 mA                       *)
(* I = 4 + (PV - PV_Min) * 16 / (PV_Max - PV_Min) *)
(* --------------------------------------------- *)

Error := FALSE;
spanPV := PV_Max - PV_Min;

IF spanPV <= 0.0 THEN
    Error := TRUE;
    I_mA := 0.0;
ELSE
    (* Wyliczenie prądu teoretycznego *)
    tmpI := 4.0 + (PV - PV_Min) * spanI / spanPV;

    IF ClampOutput THEN
        (* Ogranicz do 4–20 mA *)
        IF tmpI < 4.0 THEN
            tmpI := 4.0;
        ELSIF tmpI > 20.0 THEN
            tmpI := 20.0;
        END_IF
    END_IF

    I_mA := tmpI;
END_IF

END_FUNCTION_BLOCK

// ---- POUs/FB/FB_PressureToForce_PT1.TcPOU
FUNCTION_BLOCK FB_PressureToForce_PT1
VAR_INPUT
    Pressure_bar     : REAL;  // Ciśnienie [bar]
    PistonDiam_m     : REAL;  // Średnica tłoka [m]
    Efficiency       : REAL;  // Sprawność (0.0 .. 1.0), np. 0.9
    FilterTime_s     : REAL;  // Stała czasowa PT1 [s]
    CycleTime_s      : REAL;  // Czas cyklu PLC [s]
    EnableFilter     : BOOL;  // TRUE = filtr aktywny
    Gravity_ms2      : REAL := 9.80665; // Przysp. graw. [m/s²]
END_VAR

VAR_OUTPUT
    Force_N          : REAL;  // Siła przefiltrowana [N]
    ForceRaw_N       : REAL;  // Siła bez filtra [N]
    Force_kg         : REAL;  // Ekwiwalent masy (filtrowany) [kg]
    ForceRaw_kg      : REAL;  // Ekwiwalent masy (surowy) [kg]
END_VAR

VAR
    Pressure_Pa      : REAL;
    Area_m2          : REAL;
    Alpha            : REAL;
    ForceFilt_N      : REAL;
END_VAR

// --- Ograniczenia ---
IF Efficiency < 0.0 THEN Efficiency := 0.0; END_IF;
IF Efficiency > 1.0 THEN Efficiency := 1.0; END_IF;
IF Gravity_ms2 <= 0.0 THEN Gravity_ms2 := 9.80665; END_IF;

// --- Przeliczenia ---
Pressure_Pa := Pressure_bar * 100000.0;
Area_m2 := 3.14159265359 * (PistonDiam_m * 0.5) * (PistonDiam_m * 0.5);

// Siła surowa
ForceRaw_N := Pressure_Pa * Area_m2 * Efficiency;

// --- Filtr PT1 ---
IF EnableFilter AND (FilterTime_s > 0.0) THEN
    Alpha := CycleTime_s / FilterTime_s;
    IF Alpha > 1.0 THEN Alpha := 1.0; END_IF;

    ForceFilt_N := ForceFilt_N + Alpha * (ForceRaw_N - ForceFilt_N);
    Force_N := ForceFilt_N;
ELSE
    ForceFilt_N := ForceRaw_N;
    Force_N := ForceRaw_N;
END_IF

// --- Przeliczenie na kg ---
ForceRaw_kg := ForceRaw_N / Gravity_ms2;
Force_kg    := Force_N    / Gravity_ms2;

END_FUNCTION_BLOCK

// ---- POUs/FB/FB_ScaleTo0_10V.TcPOU
FUNCTION_BLOCK FB_ScaleTo0_10V
VAR_INPUT
    InRaw      : INT;    // Sygnał z wejścia analogowego 0–10 V (INT)
    InMin      : INT;    // Dolna granica = 0 V (np. 0)
    InMax      : INT;    // Górna granica = 10 V (np. 32767)
END_VAR
VAR_OUTPUT
    Out_V      : REAL;  // Wyjście 0–10 V
    OutPercent : REAL;  // Procent 0–100%
    Error      : BOOL;  // Błąd zakresu
END_VAR
VAR
    scaled : REAL;
END_VAR

// Zabezpieczenie przed dzieleniem przez zero
IF InMax <= InMin THEN
    Out_V := 0.0;
    OutPercent := 0.0;
    Error := TRUE;
ELSE
    Error := FALSE;
    // Konwersja INT → REAL i skalowanie do 0–1
    // Różnica w REAL, żeby InMax - InMin nie przepełniło INT
    scaled := (INT_TO_REAL(InRaw) - INT_TO_REAL(InMin)) / (INT_TO_REAL(InMax) - INT_TO_REAL(InMin));
    // Ograniczenie do 0…1
    IF scaled < 0.0 THEN scaled := 0.0; END_IF;
    IF scaled > 1.0 THEN scaled := 1.0; END_IF;
    OutPercent := scaled * 100.0;
    // Skala na 0–10 V
    Out_V := 0.0 + (scaled * 10.0);
END_IF;

END_FUNCTION_BLOCK

// ---- POUs/FB/FB_PositionOffset_4_20mA.TcPOU
FUNCTION_BLOCK FB_PositionOffset_4_20mA
VAR_INPUT
    Enable      : BOOL := TRUE;

    (* Sygnał z wejścia analogowego w mA (engineering units) *)
    In_mA        : REAL;

    (* Przycisk SET ZERO *)
    SetZero      : BOOL;

    (* Parametry liniału / skalowania *)
    Range_mm     : REAL := 125.0;   (* pełny zakres liniału *)
    mA_Min       : REAL := 4.0;
    mA_Max       : REAL := 20.0;

    (* Opcjonalnie: tolerancja do diagnostyki (np. 0.2 mA) *)
    Tol_mA       : REAL := 0.2;
END_VAR

VAR_OUTPUT
    Pos_mm           : REAL;    (* pozycja surowa 0..Range_mm *)
    PosZeroed_mm     : REAL;    (* pozycja z ofsetem (zero) *)
    Offset_mm        : REAL;    (* zapamiętany ofset *)

    InRange          : BOOL;    (* sygnał w rozsądnym zakresie *)
    UnderRange       : BOOL;    (* poniżej 4mA - Tol *)
    OverRange        : BOOL;    (* powyżej 20mA + Tol *)
END_VAR

VAR
    rTrigSetZero : R_TRIG;
    span_mA      : REAL;
    norm         : REAL;
    inClamped    : REAL;
END_VAR

(* --- wykonanie --- *)
IF NOT Enable THEN
    Pos_mm := 0.0;
    PosZeroed_mm := 0.0;
    (* Offset pozostawiamy bez zmian *)
    InRange := FALSE;
    UnderRange := FALSE;
    OverRange := FALSE;
    RETURN;
END_IF

span_mA := mA_Max - mA_Min;

(* Diagnostyka zakresu (z tolerancją) *)
UnderRange := (In_mA < (mA_Min - Tol_mA));
OverRange  := (In_mA > (mA_Max + Tol_mA));
InRange    := NOT(UnderRange OR OverRange);

(* Clamp sygnału do 4..20 mA, żeby wynik mm nie uciekał *)
inClamped := In_mA;
IF inClamped < mA_Min THEN inClamped := mA_Min; END_IF
IF inClamped > mA_Max THEN inClamped := mA_Max; END_IF

(* Skalowanie 4..20 mA -> 0..Range_mm *)
IF span_mA <= 0.0 THEN
    Pos_mm := 0.0;
ELSE
    norm := (inClamped - mA_Min) / span_mA;   (* 0..1 *)
    Pos_mm := norm * Range_mm;               (* 0..Range *)
END_IF

(* Set Zero na zboczu narastającym *)
rTrigSetZero(CLK := SetZero);
IF rTrigSetZero.Q THEN
    Offset_mm := Pos_mm;  (* zapamiętaj aktualną pozycję jako "zero" *)
END_IF

(* Pozycja z ofsetem *)
PosZeroed_mm := Pos_mm - Offset_mm;

END_FUNCTION_BLOCK

// ---- POUs/IO_Map.TcPOU
PROGRAM IO_Map
VAR
	
	
	
	AI3 AT %I*: INT;
END_VAR


//---------------------------------------------	
// EK 1818

	bControlOn				  :=  DI1_1;
	bTopPreserCmdUp           :=  DI1_2;
	bTopPreserCmdDown         :=  DI1_3;
	bCycleStartCmd            :=  DI1_4;
	bCycleStopCmd             :=  DI1_5;
	bCylinderCmdUp            :=  DI1_6;
	bCylinderCmdDown          :=  DI1_7;
	bHydraulicUnitCmdStart    :=  DI1_8;

	
	DO1_1:=bLedHydraulicUnitOn;
	DO1_2;
	DO1_3;
	DO1_4;
//--------------------------------------------	
// EL 4374	
	nHydraulicPressureRaw		:=  AI_1; //{mA]0.004=0bar/0.020=400bar
	nCylinderPositionRaw    	:=  AI_2; //[mA]0.004=0mm/0.020=125mm
	AO_1						:=nHydraulicPressureOut0_10V   	; 
	                          		AO_2;
//--------------------------------------------
	AI3;									
//--------------------------------------------
// EL 1008	
	 bHydraulicUnitRunning		:=  DI2_1;
	 bTopPreserClosed           :=  DI2_2;
	 bTopPreserMotorOk          :=  DI2_3;
	 bHydraulicUnitMotorOk      :=  DI2_4;
	 bHydraulicUnitCmdStop      :=  DI2_5;
	 bOilLevelOk                :=  DI2_6;
	 bEstopOk                   :=  DI2_7;
	                                DI2_8;
	
//--------------------------------------------
//EL 2008
	DO2_1:=bTopPreserUp ;
	DO2_2:=bTopPreserDown ;
	DO2_3:=bHydraulicUintOn ;
	DO2_4:=bLedCycleOn ;
	DO2_5:=bReliefValveOn ;
	DO2_6:=bCylinderValveUp ;
	DO2_7:=bCylinderValveDown ;
	DO2_8:=bProportionalValveEnable AND  .bCylinderValveUp ;

END_PROGRAM

// ---- POUs/BreakthroughDetection_2.TcPOU
PROGRAM BreakthroughDetection_2
VAR
	fbBreakDetect		: FB_HydraulicPress_WithBreakthroughDetection_1;
	rtAutoStart			: R_TRIG;
	rtBreak				: R_TRIG;
	fbPvTo420mA			: FB_PV_To4_20mA;
	fb4_20_to_0_10V		: FB_4_20mA_To_0_10V;
	fbDownLatch			: FB_LongPressLatch;
	TempOut				: REAL;
	bBreakDetected		: BOOL;
	rPressAtBreak		: REAL;
END_VAR


(*
	Ciśnienie albo siła wybiera GVL_ForceMode.bModeForce.
	Zakres tensometru: GVL_ForceMode.bForceRange100t (FALSE = 50 t, TRUE = 100 t).
	Napięcie celi: GVL_ForceMode.nForceInput_V, kanał 0–10 V, roboczo 0–2,5 V.

	Setpointy ciśnienia zostają na swoich wejściach.
	Drugi setpoint (siła) idzie na Force_Setpoint_*.
	Valve_Proportional wraca w barach — skalowanie 0..400 bar na 4..20 mA jest bez zmian.
*)
fbBreakDetect(
	Enable							:= bControlOn AND bEstopOk AND bCycleStopCmd,
	Mode_Manual						:= Mode.bManualMode,
	Cmd_Up_Manual					:= bCylinderCmdUp OR rtAutoStart.Q,
	Cmd_Down_Manual					:= fbDownLatch.Out,
	Pressure_Setpoint_Manual		:= GVL_HMI.nPressureSetpointManual,
	Pressure_Min_Auto				:= GVL_HMI.PressureSetpointAutoMin,
	Pressure_Max_Auto				:= GVL_HMI.PressureSetpointAutoMax,
	Position_Actual					:= Scaling.fbPos.PosZeroed_mm,
	Pressure_Actual					:= Scaling.PressureAI.PV_Value,
	Breakthrough_DeltaPress			:= GVL_HMI.nBreakDeltaPress,
	Breakthrough_DeltaPos			:= GVL_HMI.nBreakDeltaPos,
	Breakthrough_TimeWindow			:= GVL_HMI.tBreak_Time_Window,
	Ramp_Time						:= TO_TIME((GVL_HMI.nRamp_Time) * 1000),
	Mode_Force						:= GVL_ForceMode.bModeForce,
	Force_Setpoint_Manual			:= GVL_ForceMode.nForceSetpointManual,
	Force_Min_Auto					:= GVL_ForceMode.nForceSetpointAutoMin,
	Force_Max_Auto					:= GVL_ForceMode.nForceSetpointAutoMax,
	Force_Input_V					:= GVL_ForceMode.nForceInput_V,
	Force_Range_100t				:= GVL_ForceMode.bForceRange100t,
	Breakthrough_DeltaForce			:= GVL_ForceMode.nBreakDeltaForce,
	Valve_Proportional				=> TempOut,
	Coil_Up							=> bCylinderValveUp,
	Coil_Down						=> bCylinderValveDown,
	Valve_Relief					=> bReliefValveOn,
	Active							=> ,
	Auto_Active						=> bLedCycleOn,
	Breakthrough_Detected			=> bBreakDetected,
	Press_At_Break					=> rPressAtBreak,
	Pos_At_Break					=> GVL_HMI.nPositionBreak,
	Pos_At_Start					=> GVL_HMI.nPositionStart,
	Alarm							=> ,
	Force_Actual_t					=> GVL_ForceMode.nForce_t,
	Force_Actual_kg					=> GVL_ForceMode.nForce_kg,
	Force_Actual_N					=> GVL_ForceMode.nForce_N,
	Force_Actual_kN					=> GVL_ForceMode.nForce_kN,
	Force_pct						=> GVL_ForceMode.nForce_pct,
	Force_FullScale_t				=> GVL_ForceMode.nForceFullScale_t,
	Force_At_Break					=> ,
	Force_At_Break_kg				=> ,
	Force_At_Break_N				=> ,
	Force_At_Break_kN				=> ,
	Force_SensorOk					=> GVL_ForceMode.bForceSensorOk,
	Force_Overrange					=> GVL_ForceMode.bForceOverrange,
	Force_Underrange				=> GVL_ForceMode.bForceUnderrange,
	Force_SetpointLimited			=> GVL_ForceMode.bForceSetpointLimited,
	Force_CfgFault					=> GVL_ForceMode.bForceCfgFault,
	Force_Target					=> GVL_ForceMode.nForce_Target,
	Force_Setpoint_Manual_Eff		=> GVL_ForceMode.nForceSetpointManual_Eff,
	Force_Min_Auto_Eff				=> GVL_ForceMode.nForceSetpointAutoMin_Eff,
	Force_Max_Auto_Eff				=> GVL_ForceMode.nForceSetpointAutoMax_Eff,
	Breakthrough_DeltaForce_Eff		=> GVL_ForceMode.nBreakDeltaForce_Eff,
	Motion_Hold						=> GVL_ForceMode.bMotionHold);

// W trybie siły nie wpisujemy ton w pole ciśnienia przebicia.
IF NOT GVL_ForceMode.bModeForce THEN
	GVL_HMI.nPressBreak := rPressAtBreak;
END_IF

GVL_ForceMode.bForceInhibit := GVL_ForceMode.bModeForce AND NOT GVL_ForceMode.bForceSensorOk;
GVL_ForceMode.bRegulatorActive := fbBreakDetect.Active;
GVL_ForceMode.bAlarm := fbBreakDetect.Alarm OR (GVL_ForceMode.bModeForce AND GVL_ForceMode.bForceCfgFault);
IF GVL_ForceMode.bModeForce THEN
	GVL_ForceMode.nActiveSetpointManual := GVL_ForceMode.nForceSetpointManual_Eff;
	GVL_ForceMode.nActiveActual := GVL_ForceMode.nForce_t;
ELSE
	GVL_ForceMode.nActiveSetpointManual := GVL_HMI.nPressureSetpointManual;
	GVL_ForceMode.nActiveActual := Scaling.PressureAI.PV_Value;
END_IF

//============================================================
rtAutoStart(CLK:= mode.fbMode.bAutoDelayed, Q=> );
//============================================================
fbPvTo420mA(
	PV:= TempOut,
	PV_Min:= 0.0,
	PV_Max:= 400.0,
	ClampOutput:= TRUE,
	I_mA=> nHydraulicPressureOut,
	Error=> );
//=============================================================
fb4_20_to_0_10V(I_mA:= nHydraulicPressureOut, ClampOutput:= TRUE, U_V=> nHydraulicPressureOut0_10V, Error=> );
//=============================================================
fbDownLatch(
	Enable:= TRUE,
	In:= bCylinderCmdDown,
	ResetLatch:= NOT bControlOn OR NOT bEstopOk OR NOT bCycleStopCmd OR rtAutoStart.Q OR bCylinderCmdUp OR (Scaling.fbPos.PosZeroed_mm = 0) OR GVL_ForceMode.bMotionHold,
	LongTime:= T#3S,
	Out=> ,
	Latched=> );
//==============================================================
//			Siła przebicia do HMI
//==============================================================
rtBreak(CLK:= bBreakDetected, Q=> );

IF rtBreak.Q THEN
	GVL_HMI.nForce_t_Break := fbBreakDetect.Force_At_Break;
	GVL_HMI.nForce_kg_Break := fbBreakDetect.Force_At_Break_kg;
	GVL_HMI.nForce_N_Break := fbBreakDetect.Force_At_Break_N;
	GVL_HMI.nForce_kN_Break := fbBreakDetect.Force_At_Break_kN;
END_IF

IF GVL_ForceMode.bModeForce THEN
	GVL_HMI.Force_kg := GVL_ForceMode.nForce_kg;
	GVL_HMI.Force_N := GVL_ForceMode.nForce_N;
	IF rtBreak.Q THEN
		GVL_HMI.Force_kg_2 := fbBreakDetect.Force_At_Break_kg;
		GVL_HMI.Force_N_2 := fbBreakDetect.Force_At_Break_N;
	END_IF
ELSIF bBreakDetected THEN
	GVL_HMI.Force_kg_2 := GVL_HMI.Force_kg;
	GVL_HMI.Force_N_2 := GVL_HMI.Force_N;
END_IF

END_PROGRAM

// ---- POUs/FB/FB_HydraulicPress_WithBreakthroughDetection_1.TcPOU
FUNCTION_BLOCK FB_HydraulicPress_WithBreakthroughDetection_1
VAR_INPUT
    Enable              : BOOL;       // Włączenie całego układu
    Mode_Manual         : BOOL;       // TRUE = tryb ręczny, FALSE = tryb automatyczny
    Cmd_Up_Manual       : BOOL;       // Przycisk ręczny "Góra" / start AUTO
    Cmd_Down_Manual     : BOOL;       // Przycisk ręczny "Dół"

    Pressure_Setpoint_Manual : REAL; // Zadane ciśnienie w trybie ręcznym [bar]
    Pressure_Min_Auto   : REAL := 20.0;   // Ciśnienie startowe w trybie auto [bar]
    Pressure_Max_Auto   : REAL := 180.0;  // Ciśnienie docelowe w trybie auto [bar]

    Position_Actual     : REAL;       // Pozycja tłoczyska [mm]
    Pressure_Actual     : REAL;       // Ciśnienie aktualne [bar]

    // Parametry detekcji przebicia (ciśnienie)
    Breakthrough_DeltaPress : REAL := 15.0; // Spadek ciśnienia [bar]
    Breakthrough_DeltaPos   : REAL := 2.0;  // Przyrost pozycji [mm]
    Breakthrough_TimeWindow : TIME := T#150MS; // Okno czasowe analizy
    Ramp_Time                : TIME := T#10000MS; // Czas rampy AUTO min→max

    //------------------------------------------------------------------
    // Tryb siły. Domyślnie FALSE — dotychczasowe sterowanie ciśnieniem.
    //------------------------------------------------------------------
    Mode_Force               : BOOL := FALSE; // FALSE = ciśnienie, TRUE = siła
    Force_Setpoint_Manual    : REAL := 0.0;   // Drugi setpoint, ręczny [t]
    Force_Min_Auto           : REAL := 0.0;   // Siła początkowa AUTO [t]
    Force_Max_Auto           : REAL := 0.0;   // Siła docelowa AUTO [t]
    Force_Input_V            : REAL := 0.0;   // AI 0–10 V; roboczo 0–2,5 V
    Force_Range_100t         : BOOL := FALSE; // FALSE = 50 t, TRUE = 100 t
    Breakthrough_DeltaForce  : REAL := 0.0;   // Spadek siły [t]
END_VAR

VAR_OUTPUT
    Valve_Proportional  : REAL;    // Zawsze komenda zaworu w barach (0..350), nie w tonach
    Coil_Up             : BOOL;
    Coil_Down           : BOOL;
    Valve_Relief        : BOOL;    // Odciążający – otwarty gdy jest ruch w górę
    Active              : BOOL;
    Auto_Active         : BOOL;    // Czy trwa cykl automatyczny
    Breakthrough_Detected : BOOL;  // Przebicie materiału wykryte
    Press_At_Break      : REAL;    // Ciśnienie w momencie przebicia [bar]
    Pos_At_Break        : REAL;    // Pozycja w momencie przebicia
    Pos_At_Start        : REAL;    // Pozycja w momencie startu
    Alarm               : BOOL;

    Force_Actual_t      : REAL;
    Force_Actual_kg     : REAL;    // kgf
    Force_Actual_N      : REAL;
    Force_Actual_kN     : REAL;
    Force_pct           : REAL;
    Force_FullScale_t   : REAL;    // 50 albo 100
    Force_At_Break      : REAL;    // t, w chwili przebicia
    Force_At_Break_kg   : REAL;
    Force_At_Break_N    : REAL;
    Force_At_Break_kN   : REAL;
    Force_SensorOk      : BOOL;
    Force_Overrange     : BOOL;    // U > 2,55 V
    Force_Underrange    : BOOL;    // U < -0,05 V
    Force_SetpointLimited : BOOL;  // setpoint obcięty do 0..zakres albo ujemna delta
    Force_CfgFault      : BOOL;    // AutoMin > AutoMax
    Force_Target        : REAL;    // bieżące zadanie siły [t], 0 w trybie ciśnienia
    Force_Setpoint_Manual_Eff : REAL;
    Force_Min_Auto_Eff  : REAL;
    Force_Max_Auto_Eff  : REAL;
    Breakthrough_DeltaForce_Eff : REAL;
    Motion_Hold         : BOOL;    // zmiana trybu/zakresu w ruchu — puść przyciski
END_VAR

VAR
    //------------------------------------------------------------------
    // Rampa ciśnienia w AUTO – na zadany czas Ramp_Time
    //------------------------------------------------------------------
    Ramp_Timer          : TON;
    Ramp_Active         : BOOL;
    Ramp_Progress       : REAL;                  // 0.0 .. 1.0
    Pressure_Auto_Setpoint : REAL;              // Zadane ciśnienie w AUTO

    // Zmienne wewnętrzne
    State               : INT := 0;        // 0=Stop, 1=Up, 2=Down
    Pressure_Target     : REAL;
    Output_Raw          : REAL;

    // Detekcja przebicia
    Press_Prev          : REAL;
    Pos_Prev            : REAL;
    Press_Delta         : REAL;
    Pos_Delta           : REAL;
    Timer_Breakthrough  : TON;
    Breakthrough_Trigger: BOOL;

    // Zapis wartości przy przebiciu
    Press_At_Break_Int  : REAL;
    Pos_At_Break_Int    : REAL;
    Force_At_Break_Int  : REAL;

    // Do wykrywania zbocza startu AUTO
    Cmd_Up_Manual_Prev  : BOOL;
    rtAuto_Active: R_TRIG;
    fbBlink2: FB_Blink_S_1;

    // Siła
    fbForceScale        : FB_ScaleStrainGaugeForce;
    ValveCmd_Force      : REAL;     // komenda zaworu [bar] w trybie siły
    Mode_Force_Prev     : BOOL;
    Force_Range_Prev    : BOOL;
    bForceSensorFault   : BOOL;
    rPv                 : REAL;     // wielkość do detekcji: bar albo t
    rDeltaLim           : REAL;
END_VAR

// Pomiar siły. Kanał jest 0–10 V, przetwornik pracuje tylko w 0–2,5 V.
// 2,5 V = 50 t albo 100 t. Napięcie 5 V / 10 V to błąd, nie większa siła.
// Pomiar jest liczony także w trybie ciśnienia (podgląd na HMI).
//==========================================================================
fbForceScale(
    U_V         := Force_Input_V,
    Range_100t  := Force_Range_100t,
    Force_t     => Force_Actual_t,
    Force_kg    => Force_Actual_kg,
    Force_N     => Force_Actual_N,
    Force_kN    => Force_Actual_kN,
    FullScale_t => Force_FullScale_t,
    Force_pct   => Force_pct,
    SensorOk    => Force_SensorOk,
    Overrange   => Force_Overrange,
    Underrange  => Force_Underrange);

Force_SetpointLimited := FALSE;
Force_Setpoint_Manual_Eff := Force_Setpoint_Manual;
Force_Min_Auto_Eff := Force_Min_Auto;
Force_Max_Auto_Eff := Force_Max_Auto;
Breakthrough_DeltaForce_Eff := Breakthrough_DeltaForce;

IF Force_Setpoint_Manual_Eff < 0.0 THEN
    Force_Setpoint_Manual_Eff := 0.0;
    Force_SetpointLimited := TRUE;
ELSIF Force_Setpoint_Manual_Eff > Force_FullScale_t THEN
    Force_Setpoint_Manual_Eff := Force_FullScale_t;
    Force_SetpointLimited := TRUE;
END_IF

IF Force_Min_Auto_Eff < 0.0 THEN
    Force_Min_Auto_Eff := 0.0;
    Force_SetpointLimited := TRUE;
ELSIF Force_Min_Auto_Eff > Force_FullScale_t THEN
    Force_Min_Auto_Eff := Force_FullScale_t;
    Force_SetpointLimited := TRUE;
END_IF

IF Force_Max_Auto_Eff < 0.0 THEN
    Force_Max_Auto_Eff := 0.0;
    Force_SetpointLimited := TRUE;
ELSIF Force_Max_Auto_Eff > Force_FullScale_t THEN
    Force_Max_Auto_Eff := Force_FullScale_t;
    Force_SetpointLimited := TRUE;
END_IF

IF Breakthrough_DeltaForce_Eff < 0.0 THEN
    Breakthrough_DeltaForce_Eff := 0.0 - Breakthrough_DeltaForce_Eff;
    Force_SetpointLimited := TRUE;
END_IF

Force_CfgFault := Force_Min_Auto_Eff > Force_Max_Auto_Eff;
bForceSensorFault := Mode_Force AND NOT Force_SensorOk;

IF Mode_Force THEN
    rPv := Force_Actual_t;
    rDeltaLim := Breakthrough_DeltaForce_Eff;
ELSE
    rPv := Pressure_Actual;
    rDeltaLim := Breakthrough_DeltaPress;
    Force_Target := 0.0;
END_IF

//==========================================================================
// Główna logika
//==========================================================================
Active := Enable;
Breakthrough_Detected := Breakthrough_Trigger; // latch na zewnątrz

IF NOT Enable THEN
    Coil_Up := FALSE;
    Coil_Down := FALSE;
    Valve_Relief := FALSE;
    Valve_Proportional := 0.0;
    Auto_Active := FALSE;
    Alarm := FALSE;
    Breakthrough_Trigger := FALSE;
    State := 0;

    // Reset rampy
    Ramp_Active := FALSE;
    Ramp_Progress := 0.0;
    Ramp_Timer(IN := FALSE, PT := Ramp_Time);

    Cmd_Up_Manual_Prev := FALSE;
    ValveCmd_Force := 0.0;
    Motion_Hold := FALSE;
    Mode_Force_Prev := Mode_Force;
    Force_Range_Prev := Force_Range_100t;
    Force_Target := 0.0;
    RETURN;
END_IF

//------------------------------------------------------------------
// Zmiana trybu albo zakresu tensometru.
// W ruchu: postój, dopóki przyciski nie zostaną puszczone.
// Dzięki temu skok 50 t ↔ 100 t nie jest traktowany jak przebicie.
//------------------------------------------------------------------
IF (Mode_Force <> Mode_Force_Prev) OR (Force_Range_100t <> Force_Range_Prev) THEN
    IF Cmd_Up_Manual OR Cmd_Down_Manual OR Auto_Active OR (State <> 0) THEN
        Motion_Hold := TRUE;
    END_IF
    State := 0;
    Auto_Active := FALSE;
    Ramp_Active := FALSE;
    Ramp_Progress := 0.0;
    ValveCmd_Force := 0.0;
    Breakthrough_Trigger := FALSE;
    Pressure_Target := 0.0;
    Press_Prev := rPv;
    Pos_Prev := Position_Actual;
END_IF
Mode_Force_Prev := Mode_Force;
Force_Range_Prev := Force_Range_100t;

//------------------------------------------------------------------
// 1. Tryb ręczny / automatyczny
//------------------------------------------------------------------
IF Mode_Manual THEN
    // ------------------- TRYB RĘCZNY -------------------
    Auto_Active := FALSE;
    Breakthrough_Trigger := FALSE;

    IF Cmd_Up_Manual AND NOT Cmd_Down_Manual THEN
        IF bForceSensorFault THEN
            // Zły tensometr: nie budujemy siły. Dół (poniżej) zostaje dozwolony.
            State := 0;
            Pressure_Target := 0.0;
            Alarm := TRUE;
        ELSE
            State := 1;
            IF Mode_Force THEN
                // Zawór prowadzi pętla siły. Tony nie idą na wyjście proporcjonalne.
                Pressure_Target := 0.0;
            ELSE
                Pressure_Target := Pressure_Setpoint_Manual;
            END_IF
        END_IF
    ELSIF Cmd_Down_Manual AND NOT Cmd_Up_Manual THEN
        State := 2;
        Pressure_Target := 0.0;            // przy opuszczaniu zamykamy reduktor
    ELSE
        State := 0;
        Pressure_Target := 0.0;
    END_IF

    // W ręcznym rampa AUTO nieaktywna
    Ramp_Active := FALSE;
    Ramp_Progress := 0.0;
    IF NOT Mode_Force THEN
        Ramp_Timer(IN := FALSE, PT := Ramp_Time);
    END_IF

ELSE
    // ------------------- TRYB AUTOMATYCZNY -------------------
    // Start cyklu po zboczu narastającym Cmd_Up_Manual (dwuręczny / start AUTO)
    IF (Cmd_Up_Manual AND NOT Cmd_Up_Manual_Prev) AND NOT Breakthrough_Trigger THEN
        IF Mode_Force AND bForceSensorFault THEN
            Alarm := TRUE;
        ELSIF Mode_Force AND Force_CfgFault THEN
            Alarm := TRUE;
        ELSIF NOT Motion_Hold THEN
            Auto_Active := TRUE;
            State := 1;                         // jedziemy w górę

            // Start rampy
            Ramp_Active := TRUE;
            Ramp_Progress := 0.0;
            IF Mode_Force THEN
                Force_Target := Force_Min_Auto_Eff;
                ValveCmd_Force := 0.0;
            ELSE
                Pressure_Auto_Setpoint := Pressure_Min_Auto;
            END_IF
            IF NOT Mode_Force THEN
                Ramp_Timer(IN := FALSE, PT := Ramp_Time); // reset timera
            END_IF
        END_IF
    ELSE
        IF Breakthrough_Trigger OR bForceSensorFault OR (Mode_Force AND Force_CfgFault AND Auto_Active) THEN
            State := 0;                     // zatrzymujemy po przebiciu / błędzie siły
            Auto_Active := FALSE;
            Ramp_Active := FALSE;
            IF NOT Mode_Force THEN
                Ramp_Timer(IN := FALSE, PT := Ramp_Time);
            END_IF
            IF bForceSensorFault OR (Mode_Force AND Force_CfgFault) THEN
                Alarm := TRUE;
            END_IF
        END_IF
        IF NOT Mode_Force THEN
            IF Scaling.PressureAI.PV_Value>=GVL_HMI.PressureSetpointAutoMax THEN
                Ramp_Active := FALSE;
                Ramp_Timer(IN := FALSE, PT := Ramp_Time);
            END_IF
        ELSIF Force_SensorOk AND (Force_Actual_t >= Force_Max_Auto_Eff) AND (Force_Max_Auto_Eff > 0.0) THEN
            // Odpowiednik wczesnego końca rampy: siła doszła do zadania AUTO.
            Ramp_Active := FALSE;
        END_IF
    END_IF
END_IF

// Postój po zmianie trybu lub zakresu, dopóki przyciski są trzymane.
IF Motion_Hold THEN
    State := 0;
    Auto_Active := FALSE;
    Ramp_Active := FALSE;
    Pressure_Target := 0.0;
    ValveCmd_Force := 0.0;
    IF NOT Cmd_Up_Manual AND NOT Cmd_Down_Manual THEN
        Motion_Hold := FALSE;
    END_IF
END_IF

//------------------------------------------------------------------
// 2. Sterowanie kierunkiem i odciążającym
//------------------------------------------------------------------
Coil_Up   := (State = 1);
Coil_Down := (State = 2);
Valve_Relief := Coil_Up;   // zawór odciążający tylko przy ruchu w górę

//------------------------------------------------------------------
// 3. Zadane ciśnienie albo pętla siły
//    Wyjście zaworu w obu trybach jest w barach (potem 0..400 bar → 4..20 mA).
//    Krok 0,1 i sufit 350 bar są takie same jak dotychczasowy trym ciśnienia.
//------------------------------------------------------------------
IF Mode_Force THEN
    IF (State = 1) AND NOT bForceSensorFault THEN
        IF Auto_Active AND Ramp_Active THEN
            Ramp_Timer(IN := TRUE, PT := Ramp_Time);

            IF Ramp_Time > T#0s THEN
                Ramp_Progress := TIME_TO_REAL(Ramp_Timer.ET) / TIME_TO_REAL(Ramp_Time);
                IF Ramp_Progress >= 1.0 THEN
                    Ramp_Progress := 1.0;
                    Ramp_Active := FALSE;
                END_IF
            ELSE
                Ramp_Progress := 1.0;
                Ramp_Active := FALSE;
            END_IF

            Force_Target := Force_Min_Auto_Eff
                + (Force_Max_Auto_Eff - Force_Min_Auto_Eff) * Ramp_Progress;
        ELSIF Auto_Active THEN
            Force_Target := Force_Max_Auto_Eff;
            Ramp_Timer(IN := FALSE, PT := Ramp_Time);
        ELSE
            // Ręczny ruch w górę — trzymamy setpoint siły.
            Force_Target := Force_Setpoint_Manual_Eff;
            Ramp_Timer(IN := FALSE, PT := Ramp_Time);
        END_IF

        // Pętla: komenda w barach goni zmierzoną siłę do Force_Target.
        IF Force_Actual_t > Force_Target THEN
            ValveCmd_Force := ValveCmd_Force - 0.1;
        END_IF
        IF ValveCmd_Force <= 0.0 THEN
            ValveCmd_Force := 0.0;
        END_IF
        IF Force_Actual_t < Force_Target THEN
            ValveCmd_Force := ValveCmd_Force + 0.1;
        END_IF
        IF ValveCmd_Force >= 350.0 THEN
            ValveCmd_Force := 350.0;
        END_IF

        Output_Raw := ValveCmd_Force;
    ELSE
        Ramp_Timer(IN := FALSE, PT := Ramp_Time);
        Ramp_Active := FALSE;
        Ramp_Progress := 0.0;
        ValveCmd_Force := 0.0;
        Force_Target := 0.0;
        Output_Raw := 0.0;
    END_IF
ELSE
    // ------------------- TRYB CIŚNIENIA (bez zmian) -------------------
    IF Auto_Active AND State = 1 THEN
        IF Ramp_Active THEN
            // Timer rampy – pracuje tylko w czasie narastania
            Ramp_Timer(IN := TRUE, PT := Ramp_Time);

            IF Ramp_Time > T#0s THEN
                // Postęp rampy 0..1
                Ramp_Progress := TIME_TO_REAL(Ramp_Timer.ET) / TIME_TO_REAL(Ramp_Time);
                IF Ramp_Progress >= 1.0 THEN
                    Ramp_Progress := 1.0;
                    Ramp_Active := FALSE;      // rampa zakończona
                END_IF
            ELSE
                // Jeśli Ramp_Time = 0 → od razu max
                Ramp_Progress := 1.0;
                Ramp_Active := FALSE;
            END_IF

            // Liniowa rampa min→max w czasie Ramp_Time
            Pressure_Auto_Setpoint := Pressure_Min_Auto
                                    + (Pressure_Max_Auto - Pressure_Min_Auto) * Ramp_Progress;
        ELSE
            // Po zakończeniu rampy trzymamy max ciśnienie
            IF Pressure_Actual>Pressure_Max_Auto THEN
                Pressure_Auto_Setpoint:=Pressure_Auto_Setpoint-0.1;
            END_IF
            IF Pressure_Auto_Setpoint<=0 THEN
                Pressure_Auto_Setpoint:=0;
            END_IF

            IF Pressure_Actual<Pressure_Max_Auto THEN
                Pressure_Auto_Setpoint:=Pressure_Auto_Setpoint+0.1;
            END_IF
            IF Pressure_Auto_Setpoint>=350 THEN
                Pressure_Auto_Setpoint:=350;
            END_IF

            //Pressure_Auto_Setpoint := Pressure_Max_Auto;
            Ramp_Timer(IN := FALSE, PT := Ramp_Time);
        END_IF

        Output_Raw := Pressure_Auto_Setpoint;

    ELSE
        // Poza AUTO lub brak ruchu w górę – rampa nie pracuje
        Ramp_Timer(IN := FALSE, PT := Ramp_Time);
        Ramp_Active := FALSE;
        Ramp_Progress := 0.0;

        Output_Raw := Pressure_Target;
    END_IF
END_IF

// Tu możesz ewentualnie dodać LIMIT na Output_Raw → np. 0..100%
Valve_Proportional := Output_Raw;
//Valve_Proportional := LIMIT(4.0, Output_Raw, 20.0);

//------------------------------------------------------------------
// 4. Detekcja przebicia materiału
//    Ciśnienie: spadek barów. Siła: spadek ton. Pozycja jest wspólna.
//    Przy złym tensometrze w trybie siły detekcja stoi — 0 V albo 10 V
//    nie może zostać uznane za przebicie.
//------------------------------------------------------------------
IF (State = 1) AND (NOT Mode_Force OR Force_SensorOk) THEN
    Press_Delta := Press_Prev - rPv;   // spadek = dodatnia wartość
    Pos_Delta   := Position_Actual - Pos_Prev;

    IF (Press_Delta > rDeltaLim) AND (Pos_Delta > Breakthrough_DeltaPos) THEN
        Timer_Breakthrough(IN := TRUE, PT := Breakthrough_TimeWindow);
        IF Timer_Breakthrough.Q THEN
            Breakthrough_Trigger := TRUE;
            IF Mode_Force THEN
                Force_At_Break_Int := Force_Actual_t + (Press_Delta / 2.0);
            ELSE
                Press_At_Break_Int := Pressure_Actual + (Press_Delta / 2.0);
                Force_At_Break_Int := Force_Actual_t;
            END_IF
            Pos_At_Break_Int   := Position_Actual - (Pos_Delta / 2.0);
        END_IF
    ELSE
        Timer_Breakthrough(IN := FALSE);
    END_IF
ELSE
    Timer_Breakthrough(IN := FALSE);
    Breakthrough_Trigger := FALSE;   // reset przy nowym cyklu (ew. pod inny warunek)
END_IF

// Przechowanie wartości na zewnątrz
Press_At_Break := Press_At_Break_Int;
Pos_At_Break   := Pos_At_Break_Int;
Force_At_Break := Force_At_Break_Int;
Force_At_Break_kg := Force_At_Break_Int * 1000.0;
Force_At_Break_N := Force_At_Break_kg * 9.80665; // 1 kgf = 9,80665 N — to samo co FB_ScaleStrainGaugeForce
Force_At_Break_kN := Force_At_Break_N / 1000.0;

fbBlink2(Tv:= Breakthrough_TimeWindow , Q=> );///?????????????????????
// Zapis na następny cykl
IF fbBlink2.Q THEN
    Press_Prev := rPv;
    Pos_Prev   := Position_Actual;
END_IF
//------------------------------------------------------------------
// 5. Zatrzymanie po przebiciu i alarmy
//------------------------------------------------------------------
IF Breakthrough_Trigger THEN
    State := 0;
    Auto_Active := FALSE;
    Alarm := TRUE;
END_IF

//------------------------------------------------------------------
// 6. Zapamiętanie stanu przycisku (zbocze narastające)
//------------------------------------------------------------------
Cmd_Up_Manual_Prev := Cmd_Up_Manual;
//------------------------------------------------------------------
//	7.	Zapamiętanie pozycji startowej
rtAuto_Active(CLK:=Auto_Active , Q=> );

IF rtAuto_Active.Q THEN
    Pos_At_Start:=Position_Actual;
END_IF

END_FUNCTION_BLOCK

// ---- POUs/FB/FB_ScaleStrainGaugeForce.TcPOU
FUNCTION_BLOCK FB_ScaleStrainGaugeForce
VAR_INPUT
	U_V			: REAL;		(* Napięcie z kanału analogowego 0–10 V. *)
	Range_100t	: BOOL;		(* FALSE = tensometr 50 t, TRUE = tensometr 100 t. *)
END_VAR
VAR_OUTPUT
	Force_t			: REAL;	(* t (tona-siła) *)
	Force_kg		: REAL;	(* kgf *)
	Force_N			: REAL;
	Force_kN		: REAL;
	FullScale_t		: REAL;	(* 50 albo 100 *)
	Force_pct		: REAL;	(* 0–100% wybranego zakresu; przy przekroczeniu napięcia 100 i SensorOk = FALSE *)
	SensorOk		: BOOL;
	Overrange		: BOOL;	(* U > 2,55 V — nie skalujemy liniowo do 10 V *)
	Underrange		: BOOL;	(* U < -0,05 V *)
END_VAR
VAR CONSTANT
	cU_FullScale	: REAL := 2.5;		(* 2,5 V = 100% zakresu 50 t albo 100 t *)
	cU_Overrange	: REAL := 2.55;		(* zapas na szum; powyżej = błąd, nie ekstrapolacja *)
	cU_Underrange	: REAL := -0.05;
	cTonToKgf		: REAL := 1000.0;	(* 1 t = 1000 kgf *)
	cKgfToN			: REAL := 9.80665;	(* 1 kgf = 9,80665 N *)
END_VAR
VAR
	rClamped		: REAL;
END_VAR

(*
	Przetwornik tensometryczny jest podany na wejście 0–10 V,
	ale pracuje tylko w zakresie 0–2,5 V:

	    0,0 V = 0 t
	    2,5 V = 50 t  gdy Range_100t = FALSE
	    2,5 V = 100 t gdy Range_100t = TRUE

	Napięcie 5 V albo 10 V NIE oznacza wielokrotności zakresu.
	To przekroczenie (Overrange): siła do podglądu = pełny zakres, SensorOk = FALSE.
	Pasmo 2,50–2,55 V jest obcinane do 100% (szum przy pełnej skali).
	Lekki minus do -0,05 V jest zerem. Poniżej: Underrange.
*)

IF Range_100t THEN
	FullScale_t := 100.0;
ELSE
	FullScale_t := 50.0;
END_IF

Overrange := FALSE;
Underrange := FALSE;
SensorOk := FALSE;
Force_t := 0.0;
Force_pct := 0.0;
rClamped := 0.0;

IF cU_FullScale > 0.0 THEN
	Overrange := U_V > cU_Overrange;
	Underrange := U_V < cU_Underrange;

	IF Overrange THEN
		Force_t := FullScale_t;
		Force_pct := 100.0;
	ELSIF Underrange THEN
		Force_t := 0.0;
		Force_pct := 0.0;
	ELSE
		SensorOk := TRUE;
		rClamped := LIMIT(0.0, U_V, cU_FullScale);
		Force_t := (rClamped / cU_FullScale) * FullScale_t;
		Force_pct := (rClamped / cU_FullScale) * 100.0;
	END_IF
END_IF

Force_kg := Force_t * cTonToKgf;
Force_N := Force_kg * cKgfToN;
Force_kN := Force_N / 1000.0;

END_FUNCTION_BLOCK

// ---- POUs/FB/FB_4_20mA_To_0_10V.TcPOU
FUNCTION_BLOCK FB_4_20mA_To_0_10V
VAR_INPUT
    I_mA         : LREAL; (* prąd wejściowy w mA *)
    ClampOutput  : BOOL;  (* TRUE – ogranicz wyjście do 0–10 V *)
END_VAR

VAR_OUTPUT
    U_V     : LREAL; (* napięcie wyjściowe w V *)
    Error   : BOOL;  (* TRUE gdy prąd < 4 mA lub > 20 mA *)
END_VAR

VAR
    spanI  : LREAL := 16.0; (* 20 mA - 4 mA *)
    spanU  : LREAL := 10.0; (* 10 V - 0 V *)
    tmpU   : LREAL;
END_VAR

(* --------------------------------------------- *)
(* Konwersja 4–20 mA -> 0–10 V                   *)
(* U = (I - 4) * 10 / 16                         *)
(* --------------------------------------------- *)

Error := FALSE;

(* detekcja błędu zakresu *)
IF (I_mA < 4.0) OR (I_mA > 20.0) THEN
    Error := TRUE;
END_IF;

(* skalowanie *)
tmpU := (I_mA - 4.0) * spanU / spanI;

(* opcjonalne ograniczenie *)
IF ClampOutput THEN
    IF tmpU < 0.0 THEN
        tmpU := 0.0;
    ELSIF tmpU > 10.0 THEN
        tmpU := 10.0;
    END_IF;
END_IF;

U_V := tmpU;

END_FUNCTION_BLOCK

// ---- POUs/FB/FB_LongPressLatch.TcPOU
FUNCTION_BLOCK FB_LongPressLatch
VAR_INPUT
    Enable       : BOOL := TRUE;
    In           : BOOL;                 (* przycisk/wejście *)
    ResetLatch   : BOOL;                 (* dodatkowy reset zatrzasku *)
    LongTime     : TIME := T#3s;         (* próg długiego przytrzymania *)
END_VAR

VAR_OUTPUT
    Out          : BOOL;                 (* wyjście *)
    Latched      : BOOL;                 (* status zatrzasku *)
END_VAR

VAR
    tLong        : TON;
    rRiseIn      : R_TRIG;
    rFallIn      : F_TRIG;

    longReached  : BOOL;                 (* czy w tym cyklu przytrzymania osiągnięto LongTime *)
END_VAR

IF NOT Enable THEN
    Out := FALSE;
    Latched := FALSE;
    tLong(IN := FALSE, PT := LongTime);
    longReached := FALSE;
    RETURN;
END_IF

(* detekcja zboczy *)
rRiseIn(CLK := In);
rFallIn(CLK := In);

(* tLong liczy tylko gdy przycisk jest wciśnięty i NIE jesteśmy w latchu *)
tLong(IN := In AND NOT Latched, PT := LongTime);

(* dodatkowy reset zatrzasku *)
IF ResetLatch THEN
    Latched := FALSE;
END_IF

(* Jeśli jesteśmy w latchu: kolejne naciśnięcie kasuje latch *)
IF Latched AND rRiseIn.Q THEN
    Latched := FALSE;
END_IF

(* Start nowego "naciśnięcia": wyczyść longReached *)
IF rRiseIn.Q THEN
    longReached := FALSE;
END_IF

(* Osiągnięto czas długiego przytrzymania -> ustaw latch *)
IF (NOT Latched) AND tLong.Q AND (NOT longReached) THEN
    Latched := TRUE;
    longReached := TRUE;
END_IF

(* Logika wyjścia:
   - jeśli zatrzask: zawsze 1
   - jeśli nie zatrzask: wyjście jak wejście
*)
IF Latched THEN
    Out := TRUE;
ELSE
    Out := In;
END_IF

(* Po puszczeniu przycisku, jeśli nie było długiego przytrzymania,
   longReached zostaje FALSE (i tak resetujemy na kolejnym narastaniu). *)
IF rFallIn.Q THEN
    (* opcjonalnie: nic nie rób *)
END_IF

END_FUNCTION_BLOCK

// ---- POUs/Mode.TcPOU
PROGRAM Mode
VAR
	fbMode       : FB_AutoManual;
   

    bAutoMode    : BOOL;
    bManualMode  : BOOL;
    bAutoReady   : BOOL;   // np. wyjście po opóźnieniu
END_VAR

fbMode(
    bControlOn  := bControlOn,
    bEstopOK    := bEstopOK,
    bMoveUp     := .bCylinderCmdUp,
    bMoveDown   := .bCylinderCmdDown,
    bCycleStart := .bCycleStartCmd,
    bCycleStop  := .bCycleStopCmd,
    tAutoDelay  := T#1S   // np. 1 sekunda opóźnienia
);

bAutoMode   := fbMode.bAutoMode;
bManualMode := fbMode.bManualMode;
bAutoReady  := fbMode.bAutoDelayed;


IF bAutoMode THEN
	GVL_HMI.sMode:='TRYB AUTOMATYCZNY';
	ELSE
		GVL_HMI.sMode:='TRYB RĘCZNY';	
END_IF

END_PROGRAM

// ---- POUs/FB/FB_AutoManual.TcPOU
FUNCTION_BLOCK FB_AutoManual
VAR_INPUT
    bControlOn   : BOOL;   // sterownik włączony
    bEstopOK     : BOOL;   // bezpieczeństwo OK
    bMoveUp      : BOOL;   // ręczny ruch w górę
    bMoveDown    : BOOL;   // ręczny ruch w dół
    bCycleStart  : BOOL;   // start trybu auto
    bCycleStop   : BOOL;   // stop / powrót do manual
    tAutoDelay   : TIME := T#2S;   // opóźnienie wyjścia w AUTO
END_VAR

VAR_OUTPUT
    bManualMode  : BOOL;   // aktualnie MANUAL
    bAutoMode    : BOOL;   // aktualnie AUTO
    bAutoDelayed : BOOL;   // wyjście załączane z opóźnieniem po wejściu w AUTO
END_VAR

VAR
    eMode        : E_Mode := Mode_Manual;

    // detekcja zboczy
    rStart       : R_TRIG;
    rStop        : R_TRIG;
    rMoveUp      : R_TRIG;
    rMoveDown    : R_TRIG;

    // timer opóźniający wyjście w AUTO
    tonAutoDelay : TON;

    bDelayIn     : BOOL;
	//Mode_Manual: E_Mode;
	//Mode_Auto: E_Mode;
END_VAR

// ------------------------------------------------------------
// Główna logika
// ------------------------------------------------------------
bDelayIn := FALSE;  // domyślnie timer nieaktywny w tej cyklicznej iteracji

// 1. Jeśli sterowanie wyłączone lub E-STOP nie OK → zawsze MANUAL
IF NOT bControlOn OR NOT bEstopOK THEN
    eMode := Mode_Manual;
ELSE
    // 2. Detekcja zboczy przycisków
    rStart(CLK := bCycleStart);
    rStop(CLK  := NOT bCycleStop);
    rMoveUp(CLK   := bMoveUp);
    rMoveDown(CLK := bMoveDown);

    // 3. Maszyna stanów MANUAL / AUTO
    CASE eMode OF

        // ---------------- MANUAL ----------------
        0:
            // przejście do AUTO tylko na zboczu bCycleStart
            IF rStart.Q THEN
                eMode := Mode_Auto;
            END_IF;

        // ---------------- AUTO ------------------
        1:
            // każde z tych zdarzeń wraca do MANUAL:
            // - CycleStop
            // - ręczny ruch (MoveUp / MoveDown)
            // - (opcjonalnie rozbudujesz o inne warunki)
            IF rStop.Q OR rMoveUp.Q OR rMoveDown.Q THEN
                eMode := Mode_Manual;
            ELSE
                // w AUTO włączamy opóźnienie (timer)
                bDelayIn := TRUE;
            END_IF;

    END_CASE;
END_IF;

// 4. Ustawienie sygnałów trybu
bAutoMode   := (eMode = Mode_Auto);
bManualMode := NOT bAutoMode;

// 5. Obsługa timera opóźnienia wyjścia w AUTO
tonAutoDelay(
    IN := bDelayIn AND bAutoMode,  // timer działa tylko, gdy jesteśmy w AUTO
    PT := tAutoDelay
);

// wyjście opóźnione – tylko w AUTO
bAutoDelayed := tonAutoDelay.Q AND bAutoMode;

END_FUNCTION_BLOCK

// ---- POUs/POUs/Events/P_Events.TcPOU
//==================================================================================================
//							Beckhoff Automation Poland
//									23.05.2017
//	Program obslugujacy proste alarmy historyczne.
//	W opcjach wizualizacji trzeba wybrac use uniceode strings i use current visu variable
// 	v1.0	|| TC v 3.1.4020.32		|| - pierwsza wersja
//==================================================================================================
PROGRAM P_Events
VAR
	fbLocalSystemTime						: FB_LocalSystemTime;
	bEventTableSizeError					: BOOL;					// Niewlasciwy rozmiar tablicy zdarzen - sprawdz GVL_EHS.diNoOfEvents
	bEventDefinitionSizeError				: BOOL;					// Niewlasciwy rozmiar tablicy zdarzen - sprawdz GVL_EHS.diEventsDefinition
	testString: STRING(19);
END_VAR

fbLocalSystemTime(bEnable:= TRUE, systemTime=> GVL_EHS.stActTime);
//GVL_EHS.dtActTime 							:=SYSTEMTIME_TO_DT(GVL_EHS.stActTime);
GVL_EHS.dtActTime:=SYSTEMTIME_TO_STRING(in:=GVL_EHS.stActTime );
testString :=SYSTEMTIME_TO_STRING(in:=GVL_EHS.stActTime );
P_EventsDefinition ();

bEventDefinitionSizeError 					:= GVL_EHS.diEventsDefinition < 5 OR GVL_EHS.diEventsDefinition > 1000;
bEventTableSizeError 						:= GVL_EHS.diNoOfEvents < 5 OR GVL_EHS.diNoOfEvents > 1000;

IF NOT bEventDefinitionSizeError AND NOT bEventTableSizeError THEN
	IF fbLocalSystemTime.bValid THEN
		P_EventsHandling();
	END_IF
	// Visu i filtry
	P_EventsVisu();	
END_IF

P_EventHandling2();

END_PROGRAM

// ---- POUs/POUs/Events/P_EventsDefinition.TcPOU
//==================================================================================================
//							Beckhoff Automation Poland
//									23.05.2017
//	Program definiujacy zdarzenia - musi byc dostosowany do aplikacji
//	W pierwszym cyklu definiowane sa klasy
//	Zmiana jezyka na zdarzenie i w pierwszym cyklu
//	Wykrywanie aktywnosci zdarzenia i parametru - cykliczne
// 	v1.0	|| TC v 3.1.4020.32		|| - pierwsza wersja
//==================================================================================================
PROGRAM P_EventsDefinition
VAR
	bFirstCycle 							: BOOL := TRUE;
	dwPreviousLanguageID					: DWORD;
	i										: INT;
	temp: bool;
	test: BOOL;
END_VAR

// Class
IF bFirstCycle THEN
	ACT_ClassDefinition();
	bFirstCycle 							:= FALSE;
END_IF

// Language
ACT_Language();

// Active
ACT_Active();

ACTION ACT_1033_US:
// Fatal Error
GVL_EHS.arrEventDefinition[1].wsMessage	 	:= "Error01";

// Warning
GVL_EHS.arrEventDefinition[101].wsMessage 	:= "Warning01";

// Message
GVL_EHS.arrEventDefinition[201].wsMessage 	:= "Message01";
END_ACTION

ACTION ACT_1045_PL:
// Blad krytyczny
GVL_EHS.arrEventDefinition[1].wsMessage	 	:= "Hydraulika. Zabezpieczenie termiczne silnika pompy";
GVL_EHS.arrEventDefinition[2].wsMessage	 	:= "Docisk. Zabezpieczenie termiczne silnika";
GVL_EHS.arrEventDefinition[3].wsMessage	 	:= "Usterka czujnika pozycji siłownika";
GVL_EHS.arrEventDefinition[4].wsMessage	 	:= "Usterka czujnika ciśnienia";
GVL_EHS.arrEventDefinition[5].wsMessage	 	:= "";
GVL_EHS.arrEventDefinition[6].wsMessage	 	:= "";
GVL_EHS.arrEventDefinition[7].wsMessage	 	:= "";
GVL_EHS.arrEventDefinition[8].wsMessage	 	:= "";
GVL_EHS.arrEventDefinition[9].wsMessage	 	:= "";
GVL_EHS.arrEventDefinition[10].wsMessage	:= "";
GVL_EHS.arrEventDefinition[11].wsMessage	:= "";
GVL_EHS.arrEventDefinition[12].wsMessage	:= "";
GVL_EHS.arrEventDefinition[13].wsMessage	:= "";
GVL_EHS.arrEventDefinition[14].wsMessage	:= "";




// Warning
GVL_EHS.arrEventDefinition[101].wsMessage 	:= "";
GVL_EHS.arrEventDefinition[102].wsMessage 	:= "";
GVL_EHS.arrEventDefinition[103].wsMessage 	:= "";
GVL_EHS.arrEventDefinition[104].wsMessage 	:= "";
GVL_EHS.arrEventDefinition[105].wsMessage 	:= "";
GVL_EHS.arrEventDefinition[106].wsMessage   := "";
// Alarmy lekkie
GVL_EHS.arrEventDefinition[201].wsMessage 	:= "";
END_ACTION

ACTION ACT_Active:
GVL_EHS.arrEventDefinition[1].bActive:= GVL_Event.aAlarm[1];
GVL_EHS.arrEventDefinition[2].bActive:= GVL_Event.aAlarm[2];
GVL_EHS.arrEventDefinition[3].bActive:= GVL_Event.aAlarm[3];
GVL_EHS.arrEventDefinition[4].bActive:= GVL_Event.aAlarm[4];
GVL_EHS.arrEventDefinition[5].bActive:= FALSE;
GVL_EHS.arrEventDefinition[6].bActive:= FALSE;
GVL_EHS.arrEventDefinition[7].bActive:= FALSE;
GVL_EHS.arrEventDefinition[8].bActive:= FALSE;
GVL_EHS.arrEventDefinition[9].bActive:= FALSE;
GVL_EHS.arrEventDefinition[10].bActive:=FALSE;
GVL_EHS.arrEventDefinition[11].bActive:= FALSE;
GVL_EHS.arrEventDefinition[12].bActive:= FALSE;
GVL_EHS.arrEventDefinition[13].bActive:= FALSE;

GVL_EHS.arrEventDefinition[101].bActive:=FALSE;//żółte


GVL_EHS.arrEventDefinition[201].bActive:=FALSE;// zielone
END_ACTION

ACTION ACT_ClassDefinition:
FOR i := 1 TO 100 DO
	// Error - [1..100] - Class 0
	GVL_EHS.arrEventDefinition[i].dwClass := 0;
	// Warning - [101..200] - Class 1
	GVL_EHS.arrEventDefinition[100+i].dwClass := 1;
	// Message - [201..300] - Class 2
	GVL_EHS.arrEventDefinition[200+i].dwClass := 2;
END_FOR
END_ACTION

ACTION ACT_Language:
// Wybor jezyka
IF dwPreviousLanguageID <> GVL_EHS.dwLanguageId THEN
	CASE GVL_EHS.dwLanguageId OF
		
		1033:	// United States
			ACT_1033_US();
			
		1045:	// Polish
			ACT_1045_PL();
	
	ELSE	// Default Polish
		
			ACT_1045_PL();
	END_CASE
END_IF

dwPreviousLanguageID := GVL_EHS.dwLanguageId;
END_ACTION

END_PROGRAM

// ---- POUs/POUs/Events/P_EventsHandling.TcPOU
//==================================================================================================
//							Beckhoff Automation Poland
//									23.05.2017
//	Program obslugujacy zdarzenia historyczne - edycji podlega tylko tRefreshTime i bRealTime
// 	v1.0	|| TC v 3.1.4020.32		|| - pierwsza wersja
//==================================================================================================
PROGRAM P_EventsHandling
VAR
	bRealTime								: BOOL := TRUE;		// Odswiezanie ciagle - zmieniamy na FALSE tylko gdy jest duze obciazenie CPU
																// Zmiana na FLASE powoduje odfiltrowanie alarmow zgodnie z czasem tRefreshTime
	tonRefresh								: TON;				// Timer odswiezenia
	tRefreshTime							: TIME := T#1S;		// Czestotliwosc odswiezania - im dluzszy szac tym wieksze ryzyko niezauwazenia wystapienia alarmu
	bInitialized							: BOOL;				// Flaga inicjalizacji
	i										: UDINT;				// Iterator petli
	// Tablice wykrycia poczatku/konca zdarzenia
	arrSet									: ARRAY [1..GVL_EHS.diEventsDefinition] OF R_TRIG;
	arrReset								: ARRAY [1..GVL_EHS.diEventsDefinition] OF F_TRIG;
	
END_VAR

// Inicjalizacja - po uruchomieniu znajdz niezakonczone alarmy i dodaj aktualny czas jako zakonczenie
IF NOT bInitialized THEN
	FOR i := 1 TO GVL_EHS.diEventsDefinition DO
		F_RESET_Event(dwID:= i, dtActTime:= GVL_EHS.dtActTime);
	END_FOR	
	bInitialized 							:= TRUE;
END_IF

// Timer odswiezania
tonRefresh(IN:= NOT tonRefresh.Q, PT:= tRefreshTime, Q=> , ET=> );

IF bRealTime OR tonRefresh.Q THEN
	FOR i := 1 TO GVL_EHS.diEventsDefinition DO
		// Wykrycie pojawienia sie zdarzenia - ustawienie flagi na 1 cykl i dodanie na poczatek listy
		arrSet[i](CLK:= GVL_EHS.arrEventDefinition[i].bActive);
		IF arrSet[i].Q THEN
			F_SET_Event(dwID:= i, stEventDefinition:= GVL_EHS.arrEventDefinition[i], dtActTime:= GVL_EHS.dtActTime);
			
		END_IF
		// Wykrycie zakonczenia zdarzenia - ustawienie flagi na 1 cykl i dodanie daty zakonczenia
		arrReset[i](CLK:= GVL_EHS.arrEventDefinition[i].bActive);
		IF arrReset[i].Q THEN
			F_RESET_Event(dwID:= i, dtActTime:= GVL_EHS.dtActTime);
			
		END_IF
	END_FOR	
END_IF

END_PROGRAM

// ---- POUs/POUs/Events/F_RESET_Event.TcPOU
FUNCTION F_RESET_Event : BOOL
VAR_INPUT
	dwID									: DWORD;
	dtActTime								: STRING(19);//DT;
END_VAR
VAR
	i										: UDINT;
END_VAR

// Znajdz i wstaw date zakonczenia
FOR i := 1 TO GVL_EHS.diNoOfEvents DO
	IF 	GVL_EHSP.arrEvent[i].dwID = dwID THEN
		GVL_EHSP.arrEvent[i].dtDateEnd		:= dtActTime;
		EXIT;
	END_IF
END_FOR

END_FUNCTION

// ---- POUs/POUs/Events/F_SET_Event.TcPOU
FUNCTION F_SET_Event : BOOL
VAR_INPUT
	dwID									: DWORD;
	stEventDefinition						: ST_EventDefinition;
	dtActTime								: STRING(19);//DT;
END_VAR
VAR
	i										: uDINT;
END_VAR

// Przesun elemety tablicy
FOR i := 0 TO GVL_EHS.diNoOfEvents-2 DO
	GVL_EHSP.arrEvent[GVL_EHS.diNoOfEvents-i] := GVL_EHSP.arrEvent[GVL_EHS.diNoOfEvents-i-1];
END_FOR
// Dodaj nowy
GVL_EHSP.arrEvent[1].dwID					:= dwID;
GVL_EHSP.arrEvent[1].dtDateBegin 			:= dtActTime;
//GVL_EHSP.arrEvent[1].dtDateEnd	 			:= DT#1970-1-1-0:0:0;
GVL_EHSP.arrEvent[1].dtDateEnd	 			:= '';
GVL_EHSP.arrEvent[1].dwParam 				:= stEventDefinition.dwParam;
GVL_EHSP.arrEvent[1].dwClass 				:= stEventDefinition.dwClass;

END_FUNCTION

// ---- POUs/POUs/Events/P_EventsVisu.TcPOU
//==================================================================================================
//							Beckhoff Automation Poland
//									23.05.2017
//	Program obslugujacy wizualizacje VISU_EventsHistoricalSimple
//	Mozliwe filtrowanie alamow. Czestotliwosc odswiezania wplywa tylko na wyswietlanie
// 	v1.0	|| TC v 3.1.4020.32		|| - pierwsza wersja
//==================================================================================================
PROGRAM P_EventsVisu
VAR
	i										: UDINT;				// Iterator tablicy przechowywanej w pamieci
	j										: UDINT;				// Iterator tablicy wyswietlanej
	bActiveWindow							: BOOL := TRUE;		// Flaga wysietlania okna - tylko wtedy odswiezamy tablice wyswietlana
	rtPageChange							: R_TRIG;			// Wykrycie przelaczenia strony
	tonRefresh								: TON;
	tRefreshTime							: TIME := T#50MS;	// Czestotliwosc odswiezania strony
	//========================= Filtry =========================
	bRemoveFromList							: BOOL; 			// Flaga pomocnicza dla filtrow - decyduje czy element ma byc dodany na wizualizacje
	// Flagi wykonywalnosci
	bFilterID								: BOOL;
	bFilterClass							: BOOL;
	bFilterActiveOnly						: BOOL;
	// Parametry
	dwFilterID								: DWORD;	
	dwFilterClass							: DWORD;
	bFilterActiveOnly3: BOOL;
END_VAR

bActiveWindow := TRUE;//VisuElems.CURRENTVISU = 'VISU_EventsHistoricalSimple';						// Flaga wysietlania okna
rtPageChange(CLK:= bActiveWindow, Q=> );													// Wykrycie zmiany strony - jednorazowo inicjalizacja
tonRefresh(IN:= bActiveWindow AND NOT tonRefresh.Q, PT:= tRefreshTime, Q=> , ET=> );		// Timer odswiezania

IF  rtPageChange.Q OR tonRefresh.Q THEN
	// Czyszczenie tablicy
	MEMSET(ADR(GVL_EHS.arrEventVisu),0,SIZEOF(GVL_EHS.arrEventVisu));
	j := 1;
	// Filters
	//Pomocnicza dla filtrowania
	bFilterActiveOnly3:=GVL_Event.bFilterActiveOnly2 OR bFilterActiveOnly;
	//-------------------------------
	FOR i := 1 TO GVL_EHS.diNoOfEvents DO
		bRemoveFromList 								:= FALSE;
		// Jesli jest element
		IF GVL_EHSP.arrEvent[i].dwID <> 0 THEN
			bRemoveFromList								:= bFilterID AND dwFilterID <> GVL_EHSP.arrEvent[i].dwID;
			bRemoveFromList								:= bRemoveFromList OR (bFilterClass AND dwFilterClass <> GVL_EHSP.arrEvent[i].dwClass);
//			bRemoveFromList								:= bRemoveFromList OR (bFilterBeginTimeFrom AND GVL_EHSP.arrEvent[i].dtDateBegin <= dtFilterBeginTimeFrom);
//			bRemoveFromList								:= bRemoveFromList OR (bFilterBeginTimeTo AND GVL_EHSP.arrEvent[i].dtDateBegin >= dtFilterBeginTimeTo);
//			bRemoveFromList								:= bRemoveFromList OR (bFilterEndTimeFrom AND GVL_EHSP.arrEvent[i].dtDateEnd <= dtFilterEndTimeFrom);
//			bRemoveFromList								:= bRemoveFromList OR (bFilterEndTimeTo AND GVL_EHSP.arrEvent[i].dtDateEnd >= dtFilterEndTimeTo);
		//	bRemoveFromList								:= bRemoveFromList OR (bFilterActiveOnly3  AND DT#1970-1-1-0:0:0 <> GVL_EHSP.arrEvent[i].dtDateEnd);
			bRemoveFromList								:= bRemoveFromList OR (bFilterActiveOnly3  AND '' <> GVL_EHSP.arrEvent[i].dtDateEnd);
			// Analogicznie dodajemy inne filtry jesli jest taka potrzeba
			// Jesli element nie zostal usuniety przez filtr to dodajemy go do tablicy alarmow wyswietlanych
			IF NOT bRemoveFromList THEN
				GVL_EHS.arrEventVisu[j].dwID 			:= GVL_EHSP.arrEvent[i].dwID;
				GVL_EHS.arrEventVisu[j].dwClass 		:= GVL_EHSP.arrEvent[i].dwClass;
				GVL_EHS.arrEventVisu[j].wsMessage		:= GVL_EHS.arrEventDefinition[GVL_EHSP.arrEvent[i].dwID].wsMessage;
				GVL_EHS.arrEventVisu[j].dwParam 		:= GVL_EHSP.arrEvent[i].dwParam;
				GVL_EHS.arrEventVisu[j].dtDateBegin 	:= GVL_EHSP.arrEvent[i].dtDateBegin;
				GVL_EHS.arrEventVisu[j].dtDateEnd 		:= GVL_EHSP.arrEvent[i].dtDateEnd;
				IF GVL_EHS.arrEventVisu[j].dwClass=0 THEN
					GVL_EHS.arrEventVisu[j].dwColor:=16#FFFF0000;
				ELSIF GVL_EHS.arrEventVisu[j].dwClass=1 THEN
					GVL_EHS.arrEventVisu[j].dwColor:=16#FFF3F24A;
				ELSIF GVL_EHS.arrEventVisu[j].dwClass=2 THEN
					GVL_EHS.arrEventVisu[j].dwColor:=16#FFFF0000;
					//GVL_EHS.arrEventVisu[j].dwColor:=16#FF4E9640;
				END_IF
				j := j + 1;
			END_IF 
		END_IF
	END_FOR
END_IF

END_PROGRAM

// ---- POUs/POUs/Events/P_EventHandling2.TcPOU
PROGRAM P_EventHandling2
VAR
	sAktywnyEkran: STRING;
	i: INT;
	
	j: INT;
	k: INT;
	i2: INT;
	tonNieMaAlarmow: TON;
	bAlarm: BOOL;
	bOstrzezenie: BOOL;
	bAalrmLekki: BOOL;
END_VAR


//==============================================================
//		ukrywanie alarmów w stopce gdy otwarty ekran alarmów
IF GVL_HMI.hmiPanel.uiMenu=1 THEN
	
GVL_Event.bFilterActiveOnly2:=FALSE;
ELSE
	GVL_Event.bFilterActiveOnly2:=TRUE;
END_IF

//==============================================================
//     sprawdzenie czy jest alarm dla pokazania-ukrycia na stopce
//FOR i:=1 TO UDINT_TO_INT(GVL_EHS.diEventsDefinition) DO
FOR i:=1 TO 100 DO
	
	bAlarm:=GVL_EHS.arrEventDefinition[i].bActive;
	IF bAlarm THEN
		GVL_Event.bJestAalrm:=TRUE;
		EXIT;
		ELSE 
			GVL_Event.bJestAalrm:=FALSE;
		
	END_IF
	
END_FOR

FOR i2:=201 TO 300 DO
	
	bAalrmLekki:=GVL_EHS.arrEventDefinition[i2].bActive;
	IF bAalrmLekki THEN
		GVL_Event.bJestAalrmLekki:=TRUE;
		EXIT;
		ELSE 
			GVL_Event.bJestAalrmLekki:=FALSE;
	END_IF
END_FOR

FOR k:=101 TO 200 DO
	bOstrzezenie:=GVL_EHS.arrEventDefinition[k].bActive;
	IF bOstrzezenie THEN	
	GVL_Event.bJestOstrzezenie:=TRUE;
	EXIT;
		ELSE 
			GVL_Event.bJestOstrzezenie:=FALSE;
	END_IF
END_FOR
//===============================================================
//		ukrywanie alarmu na stopce
IF GVL_HMI.bResetAlarm THEN
	FOR j:=0 TO 200 DO
		GVL_Event.aAlarm[j]:=FALSE;
		GVL_Event.aWarning[j]:=FALSE;
	//	GVL_Event.aMessage[j]:=FALSE;
	END_FOR
	GVL_Event.bJestAalrm:=FALSE;
	GVL_Event.bJestAalrmLekki:=FALSE;
	GVL_Event.bJestOstrzezenie:=FALSE;
	//GVL_HMI.bResetAlarm:=FALSE;
END_IF

tonNieMaAlarmow(IN:=GVL_HMI.bResetAlarm , PT:=T#500MS , Q=> , ET=> );
IF tonNieMaAlarmow.Q THEN
	GVL_HMI.bResetAlarm:=FALSE;
END_IF

END_PROGRAM

// ---- POUs/Alarms.TcPOU
PROGRAM Alarms
VAR
END_VAR


//
IF  HydraulicPump.fbHydPump.bFaultThermal THEN
	GVL_Event.aAlarm[1]:=TRUE;
	END_IF
	
IF  UpperPreserDrive.fbUupperPreser.bFault THEN
	GVL_Event.aAlarm[2]:=TRUE;
	END_IF
	
IF Scaling.fbPos.OverRange OR Scaling.fbPos.UnderRange THEN
	GVL_Event.aAlarm[3]:=TRUE;
	END_IF
	
IF NOT.Scaling.PressureAI.Valid THEN
	GVL_Event.aAlarm[4]:=TRUE;
	END_IF

END_PROGRAM

// ---- POUs/SavePresistent.TcPOU
PROGRAM SavePresistent
VAR
	fbZapisZmiennychPresistent: FB_WritePersistentData;
END_VAR

fbZapisZmiennychPresistent(
	NETID:= , 
	PORT:=851, 
	START:= .bEstopOk OR .bCycleStartCmd OR .bCycleStopCmd OR .bControlOn, 
	TMOUT:=T#2000MS , 
	MODE:=SPDM_2PASS , 
	BUSY=> , 
	ERR=> , 
	ERRID=> );

END_PROGRAM

// ---- HMI/FB/HMI.TcPOU
FUNCTION_BLOCK HMI
VAR_INPUT
	idAmsNetID  	: T_AmsNetId;
	sRecipePath		: STRING(512);
	sNazwaSzablonu	: T_MaxString;
END_VAR
VAR
	
	bTemp			: BOOL;
	bInicjacjaOK	: BOOL := FALSE;
	
	bReset			: BOOL;
	bResetMenu 		: BOOL := FALSE;

	uiMenu			: UINT := 0;
	
	arrButtony		: ARRAY[0..ILOSC_BUTTONY_MENU] OF stButton;
	
	

	bLogInBrak 		: BOOL;//:=TRUE;


	
END_VAR
VAR CONSTANT
	ILOSC_BUTTONY_MENU			: UINT := 8;  // o jeden mniej bo 0 ;
	MAX_ILOSC_ALARMY			: UINT := 100;
	MAX_ILOSC_ALARMY_NAZWY		: UINT := 20;
END_VAR




VAR_OUTPUT
	uiNumerEkranu: UINT;
END_VAR





IF NOT bInicjacjaOK THEN
	Inicjacja();
END_IF

Logowanie();
(*ObslugaReceptur();
IF bReset THEN
	IF Reset() THEN
		bReset := FALSE;
	END_IF
END_IF
*)
IF bResetMenu THEN
	IF MenuReset() THEN
		bResetMenu := FALSE;
	END_IF
END_IF
uiNumerEkranu:=uiMenu;

METHOD Inicjacja : BOOL
VAR
   	uiLicznik		: UINT;
END_VAR
VAR_INST

	
END_VAR


FOR uiLicznik := 0 TO  ILOSC_BUTTONY_MENU DO
	arrButtony[uiLicznik].bVisable 			:= FALSE;
	arrButtony[uiLicznik].bToggleCollor 	:= FALSE;
	arrButtony[uiLicznik].dwAlarmColor  	:= 16#FFABA494;
	arrButtony[uiLicznik].dwColor			:= 16#FFC0C0C0;
	arrButtony[uiLicznik].nIndexDynamicText	:= uiLicznik;
	
END_FOR

uiMenu := 0;
arrButtony[0].bToggleCollor := TRUE;
bInicjacjaOK := TRUE;
END_METHOD

METHOD Logowanie : BOOL
VAR_INPUT
END_VAR
VAR

END_VAR
VAR_INST
	fbGetCurTaskIndex 	: GETCURTASKINDEX;
	pClient				: POINTER TO VisuElems.VisuStructClientData; 
	sCurrentUser		: WSTRING :="";
	rtrigGrzyb			: R_TRIG;
	tonGrzyb			: TON;
	tonStart			: TON;
	rtrigPrzycisk3		: R_TRIG;
	rtrigPrzycisk7		: R_TRIG;
	ftrigPrzycisk3		: F_TRIG;
	ftrigPrzycisk7		: F_TRIG;
	bPrzycisk3Trwa		: BOOL;
	bPrzycisk7Trwa		: BOOL;
	
	bGrzybTrwa			: BOOL:=FALSE;
	bOpoznienieStart	: BOOL;
	
END_VAR
(*  Auto logowanie z opóźnieniem po starcie HMI
fbGetCurTaskIndex();
IF _TaskInfo[fbGetCurTaskIndex.index].FirstCycle THEN
	bOpoznienieStart := TRUE;
END_IF

tonStart(IN:=bOpoznienieStart ,PT:=T#1S);
IF tonStart.Q THEN
	bOpoznienieStart:=FALSE;
	bLogInBrak 		:= TRUE;
END_IF
*)

(*  Auto Logowanie po naciśnięciu grzyba 
rtrigGrzyb(CLK:=GVL_Inputs.bGrzybCP3916 AND NOT bOpoznienieStart);
IF rtrigGrzyb.Q THEN
	bGrzybTrwa:= TRUE;
END_IF
IF NOT GVL_Inputs.bGrzybCP3916  THEN
	bGrzybTrwa := FALSE;
END_IF

tonGrzyb(IN := bGrzybTrwa , PT:=T#1M);//5M
IF tonGrzyb.Q THEN
	bLogInBrak := TRUE;
	bGrzybTrwa := FALSE;
END_IF
*)

(* Auto logowanie po przyciśnięciu odpowiednich klawiszy
rtrigPrzycisk3( CLK:= bPrzycisk3Panel);
rtrigPrzycisk7( CLK:= bPrzycisk7Panel);
ftrigPrzycisk3( CLK:= bPrzycisk3Panel);
ftrigPrzycisk7( CLK:= bPrzycisk7Panel);

IF rtrigPrzycisk3.Q  THEN
	bPrzycisk3Trwa := TRUE;
END_IF
IF rtrigPrzycisk7.Q  THEN
	bPrzycisk7Trwa := TRUE;
END_IF
IF ftrigPrzycisk3.Q  THEN
	bPrzycisk3Trwa := FALSE;
END_IF
IF ftrigPrzycisk7.Q  THEN
	bPrzycisk7Trwa := FALSE;
END_IF

IF bPrzycisk3Trwa AND bPrzycisk7Trwa THEN
	VisuElems.g_ClientManager.BeginIteration(); 
	pClient := VisuElems.g_ClientManager.GetNextClient(); 
	WHILE pClient <> VisuElems.NULL DO 
		VisuUserManagement.g_VisuUserMgmt2.LoginToUserGroup(pClient, 2, "user", "user");
		uiMenu := 0;
		pClient := VisuElems.g_ClientManager.GetNextClient(); 
	END_WHILE

	IF sCurrentUser="brak" THEN
		bLogInBrak:=FALSE;
	END_IF

END_IF
*)

sCurrentUser:=VisuElemsWinControls.CurrentUserName;

IF bLogInBrak THEN

	VisuElems.g_ClientManager.BeginIteration(); 
	pClient := VisuElems.g_ClientManager.GetNextClient(); 
	WHILE pClient <> VisuElems.NULL DO 
		VisuUserManagement.g_VisuUserMgmt2.LoginToUserGroup(pClient, 3, "brak", "brak");
		uiMenu := 0;
		pClient := VisuElems.g_ClientManager.GetNextClient(); 
	END_WHILE

	IF sCurrentUser="brak" THEN
		bLogInBrak:=FALSE;
	END_IF

END_IF
END_METHOD

METHOD MenuReset : BOOL
VAR
   	uiLicznik		: UINT;
	
END_VAR
//usuwa podświetlenie ze wszystkich przycisków menu ale pozostawia na wybranym
FOR uiLicznik := 0 TO  ILOSC_BUTTONY_MENU DO
	arrButtony[uiLicznik].bToggleCollor := FALSE;
END_FOR
arrButtony[uiMenu].bToggleCollor := TRUE;
MenuReset := TRUE;
END_METHOD

END_FUNCTION_BLOCK

// ---- HMI/FB/FB_Blink_S.TcPOU
(********************************************************************************************)
(*							Beckhoff Automation Poland										*)
(*								FB_Blink_S	 v1.1											*)
(*									9.11.2007												*)
(*						Blok funkcyjny zegara synchronicznego								*)
(*__________________________________________________________________________________________*)

FUNCTION_BLOCK FB_Blink_S
VAR_INPUT
	Tv										:	TIME;				(*Czas trwania impulsu i przerwy*)
END_VAR
VAR_OUTPUT
	Q										:	BOOL;				(*Wyjscie*)
END_VAR
VAR
	ton1									:	TON;
	ton2									:	TON;
END_VAR

ton1(IN:= NOT ton2.Q, PT:=Tv);
Q:=ton1.Q;
ton2(IN:=ton1.Q , PT:=ton1.PT );

END_FUNCTION_BLOCK

// ---- POUs/FB/FB_AI_mA_To_mm_Adv.TcPOU
FUNCTION_BLOCK FB_AI_mA_To_mm_Adv
VAR_INPUT
    // Wejście prądowe (już w mA)
    In_mA        : REAL;       // np. 4.0 ... 20.0 mA
    InMin_mA     : REAL := 4.0;
    InMax_mA     : REAL := 20.0;

    // Zakres mechaniczny w mm
    MM_Min       : REAL;       // np. 0.0 mm
    MM_Max       : REAL;       // np. 1000.0 mm

    // Progi diagnostyczne
    LowLimit_mA  : REAL := 3.6;
    HighLimit_mA : REAL := 21.0;
END_VAR

VAR_OUTPUT
    Out_mA       : REAL;        // prąd wejściowy (przepisany)
    MM_Value     : REAL;        // pozycja w mm
    MM_Percent   : REAL;        // 0–100 %
    Status       : E_AI_Status;
    Valid        : BOOL;
END_VAR

VAR
    ratioRaw, ratioClamped : REAL;
END_VAR

// ---- Sprawdzenie poprawności konfiguracji ----
IF InMax_mA <= InMin_mA THEN
    Status      := AI_Status_ConfigError;
    Valid       := FALSE;
    Out_mA      := InMin_mA;
    MM_Value    := MM_Min;
    MM_Percent  := 0.0;
ELSE
    // ---- Krok 1: mA → udział 0..1 (bez ograniczania) ----
    ratioRaw := (In_mA - InMin_mA) / (InMax_mA - InMin_mA);

    // ---- Krok 2: diagnostyka na surowym prądzie ----
    Out_mA := In_mA;

    IF Out_mA < LowLimit_mA THEN
        Status := AI_Status_UnderRange;
        Valid  := FALSE;
    ELSIF Out_mA > HighLimit_mA THEN
        Status := AI_Status_OverRange;
        Valid  := FALSE;
    ELSE
        Status := AI_Status_Ok;
        Valid  := TRUE;
    END_IF;

    // ---- Krok 3: zacięcie udziału 0..1 ----
    ratioClamped := ratioRaw;
    IF ratioClamped < 0.0 THEN ratioClamped := 0.0; END_IF;
    IF ratioClamped > 1.0 THEN ratioClamped := 1.0; END_IF;

    // ---- Krok 4: 0..1 → mm ----
    MM_Value   := MM_Min + ratioClamped * (MM_Max - MM_Min);
    MM_Percent := ratioClamped * 100.0;
END_IF;

END_FUNCTION_BLOCK

// ---- POUs/FB/FB_HydraulicPress_Atos_420mA.TcPOU

FUNCTION_BLOCK FB_HydraulicPress_Atos_420mA
// ===============================================
//  Prasa / stanowisko wytrzymałościowe
//  Enkoder 4-20mA + zawór Atos + E-BM-AS-PS-01H/I
//  Bez zewnętrznych bibliotek – działa wszędzie
// ===============================================

VAR_INPUT
    Enable                  : BOOL := FALSE;      // Włączenie całego układu
    Mode_Manual             : BOOL := TRUE;       // TRUE = ręczny, FALSE = auto
    Cmd_Up                  : BOOL := FALSE;      // Start / góra (dwuręczny w auto)
    Cmd_Down                : BOOL := FALSE;      // Ręczny dół

